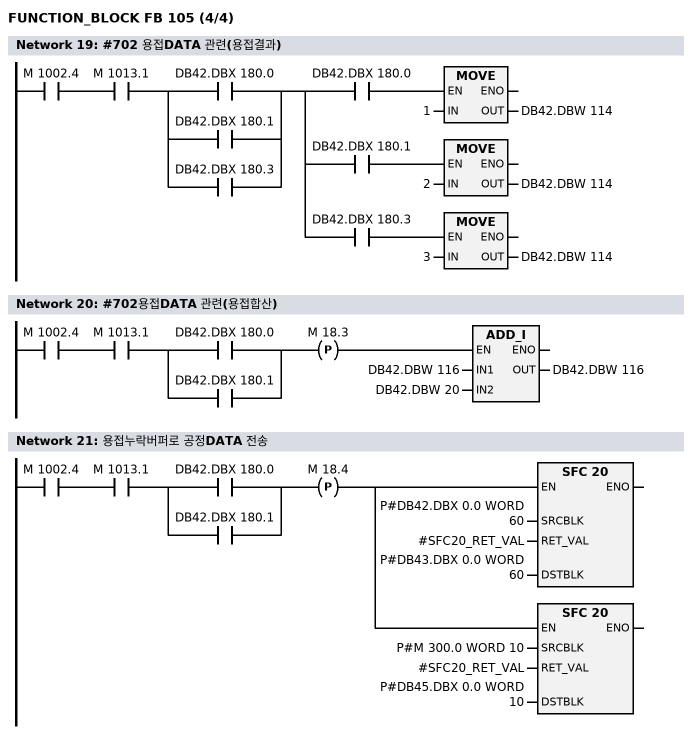

      A     M   1002.4;
      A     M   1013.1;
      A(    ;
      O     DB42.DBX  180.0;
      O     DB42.DBX  180.1;
      O     DB42.DBX  180.3;
      )     ;
      =     L      2.0;
      A     L      2.0;
      A     DB42.DBX  180.0;
      JNB   _022;
      L     1;
      T     DB42.DBW  114;
_022: NOP   0;
      A     L      2.0;
      A     DB42.DBX  180.1;
      JNB   _023;
      L     2;
      T     DB42.DBW  114;
_023: NOP   0;
      A     L      2.0;
      A     DB42.DBX  180.3;
      JNB   _024;
      L     3;
      T     DB42.DBW  114;
_024: NOP   0;
NETWORK
TITLE =#702용접DATA 관련(용접합산)

      A     M   1002.4;
      A     M   1013.1;
      A(    ;
      O     DB42.DBX  180.0;
      O     DB42.DBX  180.1;
      )     ;
      FP    M     18.3;
      JNB   _025;
      L     DB42.DBW  116;
      L     DB42.DBW   20;
      +I    ;
      T     DB42.DBW  116;
_025: NOP   0;
NETWORK
TITLE =용접누락버퍼로 공정DATA 전송

      A     M   1002.4;
      A     M   1013.1;
      A(    ;
      O     DB42.DBX  180.0;
      O     DB42.DBX  180.1;
      )     ;
      FP    M     18.4;
      =     L      2.0;
      A     L      2.0;
      JNB   _026;
      CALL SFC   20 (
           SRCBLK                   := P#DB42.DBX 0.0 WORD 60,
           RET_VAL                  := #SFC20_RET_VAL,
           DSTBLK                   := P#DB43.DBX 0.0 WORD 60);
_026: NOP   0;
      A     L      2.0;
      JNB   _027;
      CALL SFC   20 (
           SRCBLK                   := P#M 300.0 WORD 10,
           RET_VAL                  := #SFC20_RET_VAL,
           DSTBLK                   := P#DB45.DBX 0.0 WORD 10);
_027: NOP   0;
NETWORK
TITLE =용접누락버퍼로 공정DATA 전송

      A     M    501.0;
      FP    M     18.5;
      =     L      2.0;
      A(    ;
      A     L      2.0;
      JNB   _028;
      CALL SFC   20 (
           SRCBLK                   := P#DB43.DBX 960.0 WORD 60,
           RET_VAL                  := #SFC20_RET_VAL,
           DSTBLK                   := P#DB43.DBX 1080.0 WORD 60);
_028: A     BR;
      )     ;
      JNB   _029;
      CALL SFC   20 (
           SRCBLK                   := P#DB43.DBX 840.0 WORD 60,
           RET_VAL                  := #SFC20_RET_VAL,
           DSTBLK                   := P#DB43.DBX 960.0 WORD 60);
_029: NOP   0;
      A(    ;
      A     L      2.0;
      JNB   _02a;
      CALL SFC   20 (
           SRCBLK                   := P#DB43.DBX 720.0 WORD 60,
           RET_VAL                  := #SFC20_RET_VAL,
           DSTBLK                   := P#DB43.DBX 840.0 WORD 60);
_02a: A     BR;
      )     ;
      JNB   _02b;
      CALL SFC   20 (
           SRCBLK                   := P#DB43.DBX 600.0 WORD 60,
           RET_VAL                  := #SFC20_RET_VAL,
           DSTBLK                   := P#DB43.DBX 720.0 WORD 60);
_02b: NOP   0;
      A(    ;
      A     L      2.0;
      JNB   _02c;
      CALL SFC   20 (
           SRCBLK                   := P#DB43.DBX 480.0 WORD 60,
           RET_VAL                  := #SFC20_RET_VAL,
           DSTBLK                   := P#DB43.DBX 600.0 WORD 60);
_02c: A     BR;
      )     ;
      JNB   _02d;
      CALL SFC   20 (
           SRCBLK                   := P#DB43.DBX 360.0 WORD 60,
           RET_VAL                  := #SFC20_RET_VAL,
           DSTBLK                   := P#DB43.DBX 480.0 WORD 60);
_02d: NOP   0;
      A(    ;
      A     L      2.0;
      JNB   _02e;
      CALL SFC   20 (
           SRCBLK                   := P#DB43.DBX 240.0 WORD 60,
           RET_VAL                  := #SFC20_RET_VAL,
           DSTBLK                   := P#DB43.DBX 360.0 WORD 60);
_02e: A     BR;
      )     ;
      JNB   _02f;
      CALL SFC   20 (
           SRCBLK                   := P#DB43.DBX 120.0 WORD 60,
           RET_VAL                  := #SFC20_RET_VAL,
           DSTBLK                   := P#DB43.DBX 240.0 WORD 60);
_02f: NOP   0;
      A     L      2.0;
      JNB   _030;
      CALL SFC   20 (
           SRCBLK                   := P#DB43.DBX 0.0 WORD 60,
           RET_VAL                  := #SFC20_RET_VAL,
           DSTBLK                   := P#DB43.DBX 120.0 WORD 60);
_030: NOP   0;
      A     L      2.0;
      JNB   _031;
      CALL SFC   21 (
           BVAL                     := P#M 40.0 WORD 1,
           RET_VAL                  := #SFC20_RET_VAL,
           BLK                      := P#DB43.DBX 0.0 WORD 60);
_031: NOP   0;
      A(    ;
      A     L      2.0;
      JNB   _032;
      CALL SFC   20 (
           SRCBLK                   := P#DB45.DBX 160.0 WORD 10,
           RET_VAL                  := #SFC20_RET_VAL,
           DSTBLK                   := P#DB45.DBX 180.0 WORD 10);
_032: A     BR;
      )     ;
      JNB   _033;
      CALL SFC   20 (
           SRCBLK                   := P#DB45.DBX 140.0 WORD 10,
           RET_VAL                  := #SFC20_RET_VAL,
           DSTBLK                   := P#DB45.DBX 160.0 WORD 10);
_033: NOP   0;
      A(    ;
      A     L      2.0;
      JNB   _034;
      CALL SFC   20 (
           SRCBLK                   := P#DB45.DBX 120.0 WORD 10,
           RET_VAL                  := #SFC20_RET_VAL,
           DSTBLK                   := P#DB45.DBX 140.0 WORD 10);
_034: A     BR;
      )     ;
      JNB   _035;
      CALL SFC   20 (
           SRCBLK                   := P#DB45.DBX 100.0 WORD 10,
           RET_VAL                  := #SFC20_RET_VAL,
           DSTBLK                   := P#DB45.DBX 120.0 WORD 10);
_035: NOP   0;
      A(    ;
      A     L      2.0;
      JNB   _036;
      CALL SFC   20 (
           SRCBLK                   := P#DB45.DBX 80.0 WORD 10,
           RET_VAL                  := #SFC20_RET_VAL,
           DSTBLK                   := P#DB45.DBX 100.0 WORD 10);
_036: A     BR;
      )     ;
      JNB   _037;
      CALL SFC   20 (
           SRCBLK                   := P#DB45.DBX 60.0 WORD 10,
           RET_VAL                  := #SFC20_RET_VAL,
           DSTBLK                   := P#DB45.DBX 80.0 WORD 10);
_037: NOP   0;
      A(    ;
      A     L      2.0;
      JNB   _038;
      CALL SFC   20 (
           SRCBLK                   := P#DB45.DBX 40.0 WORD 10,
           RET_VAL                  := #SFC20_RET_VAL,
           DSTBLK                   := P#DB45.DBX 60.0 WORD 10);
_038: A     BR;
      )     ;
      JNB   _039;
      CALL SFC   20 (
           SRCBLK                   := P#DB45.DBX 20.0 WORD 10,
           RET_VAL                  := #SFC20_RET_VAL,
           DSTBLK                   := P#DB45.DBX 40.0 WORD 10);
_039: NOP   0;
      A     L      2.0;
      JNB   _03a;
      CALL SFC   20 (
           SRCBLK                   := P#DB45.DBX 0.0 WORD 10,
           RET_VAL                  := #SFC20_RET_VAL,
           DSTBLK                   := P#DB45.DBX 20.0 WORD 10);
_03a: NOP   0;
      A     L      2.0;
      JNB   _03b;
      CALL SFC   21 (
           BVAL                     := P#M 40.0 WORD 1,
           RET_VAL                  := #SFC20_RET_VAL,
           BLK                      := P#DB45.DBX 0.0 WORD 10);
_03b: NOP   0;
NETWORK
TITLE =용접누락버퍼로 공정DATA 전송
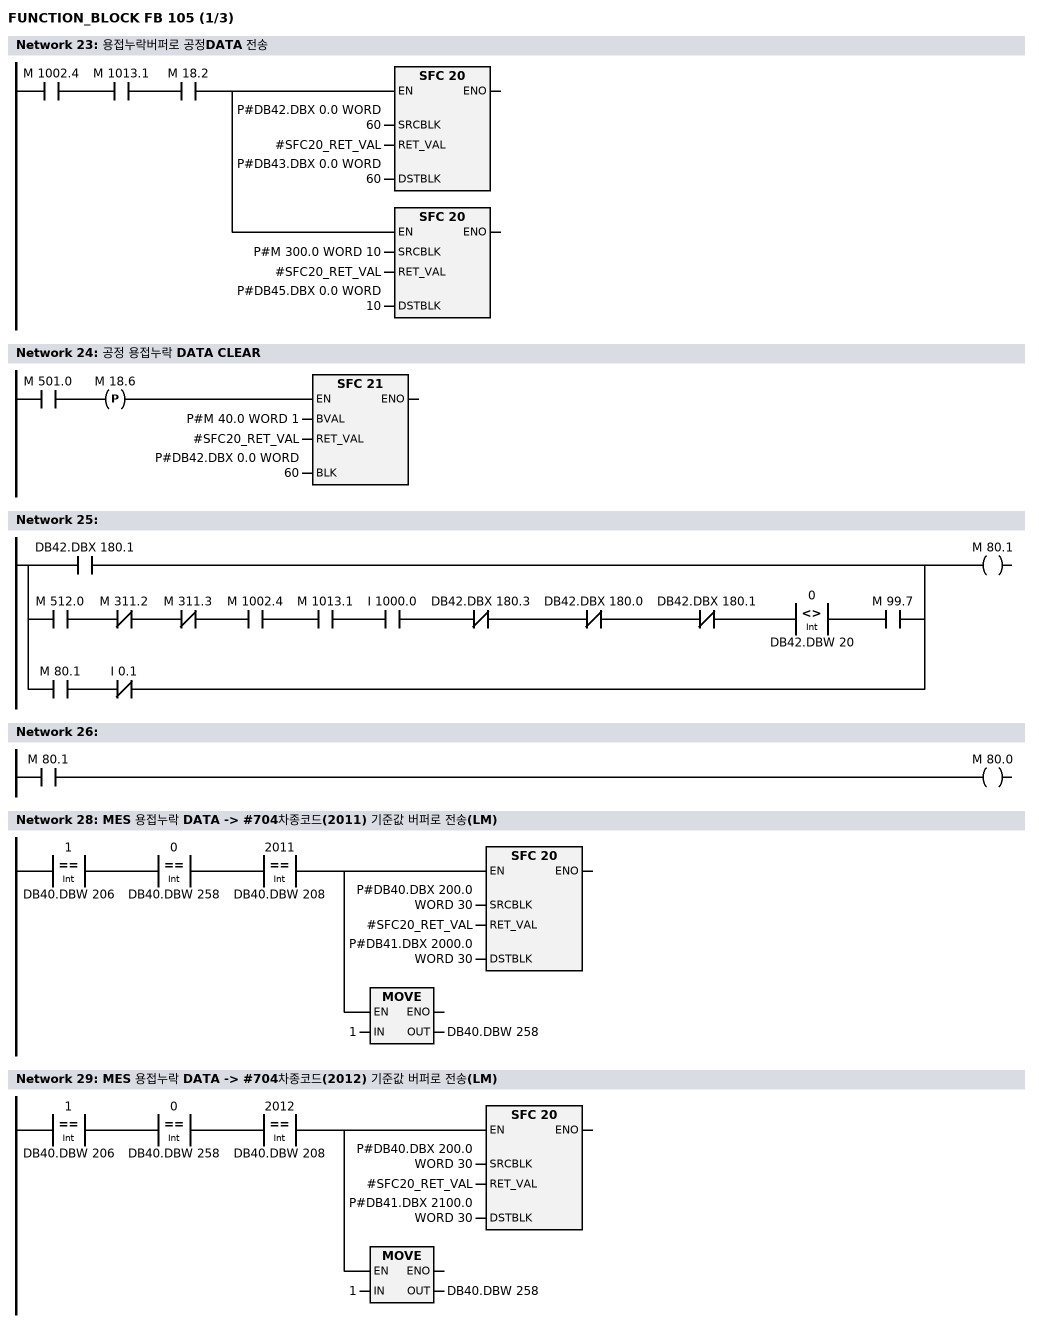

      A     M   1002.4;
      A     M   1013.1;
      A     M     18.2;
      =     L      2.0;
      A     L      2.0;
      JNB   _03c;
      CALL SFC   20 (
           SRCBLK                   := P#DB42.DBX 0.0 WORD 60,
           RET_VAL                  := #SFC20_RET_VAL,
           DSTBLK                   := P#DB43.DBX 0.0 WORD 60);
_03c: NOP   0;
      A     L      2.0;
      JNB   _03d;
      CALL SFC   20 (
           SRCBLK                   := P#M 300.0 WORD 10,
           RET_VAL                  := #SFC20_RET_VAL,
           DSTBLK                   := P#DB45.DBX 0.0 WORD 10);
_03d: NOP   0;
NETWORK
TITLE =공정 용접누락 DATA CLEAR

      A     M    501.0;
      FP    M     18.6;
      JNB   _03e;
      CALL SFC   21 (
           BVAL                     := P#M 40.0 WORD 1,
           RET_VAL                  := #SFC20_RET_VAL,
           BLK                      := P#DB42.DBX 0.0 WORD 60);
_03e: NOP   0;
NETWORK
TITLE =

      O     DB42.DBX  180.1;
      O     ;
      A     M    512.0;
      AN    M    311.2;
      AN    M    311.3;
      A     M   1002.4;
      A     M   1013.1;
      A     I   1000.0;
      AN    DB42.DBX  180.3;
      AN    DB42.DBX  180.0;
      AN    DB42.DBX  180.1;
      A(    ;
      L     0;
      L     DB42.DBW   20;
      <>I   ;
      )     ;
      A     M     99.7;
      O     ;
      A     M     80.1;
      AN    I      0.1;
      =     M     80.1;
NETWORK
TITLE =

      A     M     80.1;
      =     M     80.0;
NETWORK
TITLE =

NETWORK
TITLE =MES 용접누락 DATA -> #704차종코드(2011) 기준값 버퍼로 전송(LM)

      A(    ;
      L     1;
      L     DB40.DBW  206;
      ==I   ;
      )     ;
      A(    ;
      L     0;
      L     DB40.DBW  258;
      ==I   ;
      )     ;
      A(    ;
      L     2011;
      L     DB40.DBW  208;
      ==I   ;
      )     ;
      =     L      2.0;
      A     L      2.0;
      JNB   _03f;
      CALL SFC   20 (
           SRCBLK                   := P#DB40.DBX 200.0 WORD 30,
           RET_VAL                  := #SFC20_RET_VAL,
           DSTBLK                   := P#DB41.DBX 2000.0 WORD 30);
_03f: NOP   0;
      A     L      2.0;
      JNB   _040;
      L     1;
      T     DB40.DBW  258;
_040: NOP   0;
NETWORK
TITLE =MES 용접누락 DATA -> #704차종코드(2012) 기준값 버퍼로 전송(LM)

      A(    ;
      L     1;
      L     DB40.DBW  206;
      ==I   ;
      )     ;
      A(    ;
      L     0;
      L     DB40.DBW  258;
      ==I   ;
      )     ;
      A(    ;
      L     2012;
      L     DB40.DBW  208;
      ==I   ;
      )     ;
      =     L      2.0;
      A     L      2.0;
      JNB   _041;
      CALL SFC   20 (
           SRCBLK                   := P#DB40.DBX 200.0 WORD 30,
           RET_VAL                  := #SFC20_RET_VAL,
           DSTBLK                   := P#DB41.DBX 2100.0 WORD 30);
_041: NOP   0;
      A     L      2.0;
      JNB   _042;
      L     1;
      T     DB40.DBW  258;
_042: NOP   0;
NETWORK
TITLE =MES 용접누락 DATA -> #704차종코드(2013) 기준값 버퍼로 전송(LM)
//
//
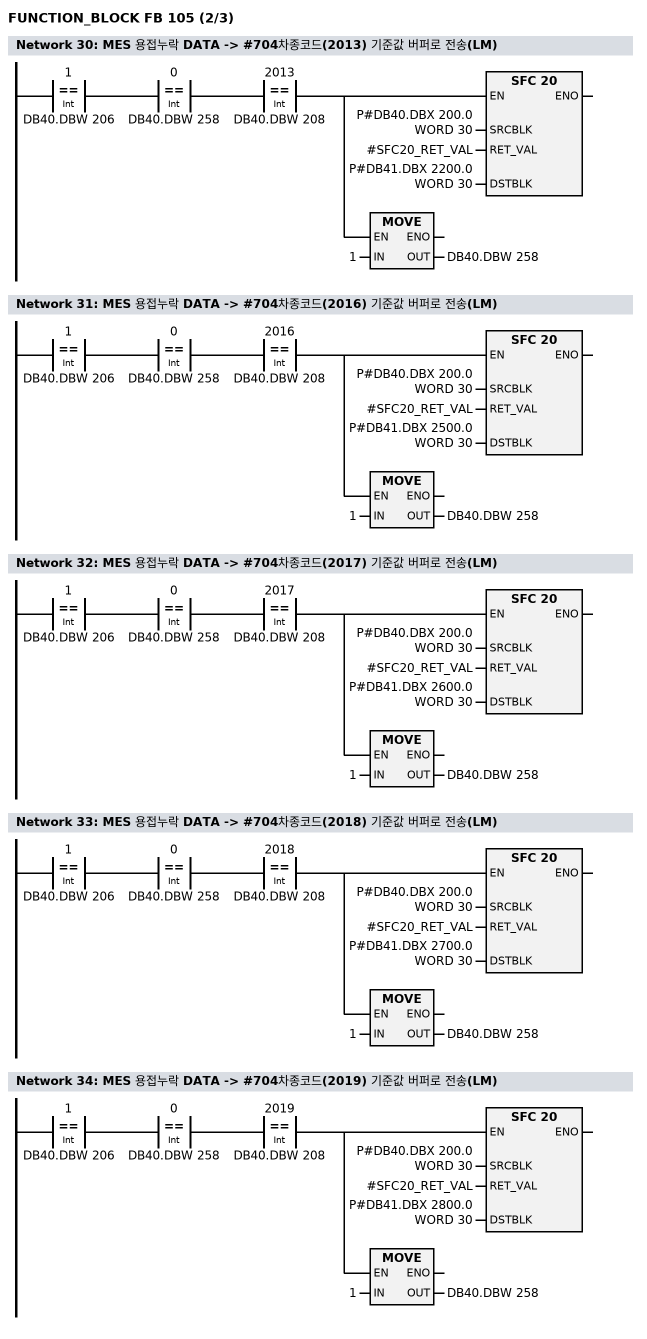
      A(    ;
      L     1;
      L     DB40.DBW  206;
      ==I   ;
      )     ;
      A(    ;
      L     0;
      L     DB40.DBW  258;
      ==I   ;
      )     ;
      A(    ;
      L     2013;
      L     DB40.DBW  208;
      ==I   ;
      )     ;
      =     L      2.0;
      A     L      2.0;
      JNB   _043;
      CALL SFC   20 (
           SRCBLK                   := P#DB40.DBX 200.0 WORD 30,
           RET_VAL                  := #SFC20_RET_VAL,
           DSTBLK                   := P#DB41.DBX 2200.0 WORD 30);
_043: NOP   0;
      A     L      2.0;
      JNB   _044;
      L     1;
      T     DB40.DBW  258;
_044: NOP   0;
NETWORK
TITLE =MES 용접누락 DATA -> #704차종코드(2016) 기준값 버퍼로 전송(LM)

      A(    ;
      L     1;
      L     DB40.DBW  206;
      ==I   ;
      )     ;
      A(    ;
      L     0;
      L     DB40.DBW  258;
      ==I   ;
      )     ;
      A(    ;
      L     2016;
      L     DB40.DBW  208;
      ==I   ;
      )     ;
      =     L      2.0;
      A     L      2.0;
      JNB   _045;
      CALL SFC   20 (
           SRCBLK                   := P#DB40.DBX 200.0 WORD 30,
           RET_VAL                  := #SFC20_RET_VAL,
           DSTBLK                   := P#DB41.DBX 2500.0 WORD 30);
_045: NOP   0;
      A     L      2.0;
      JNB   _046;
      L     1;
      T     DB40.DBW  258;
_046: NOP   0;
NETWORK
TITLE =MES 용접누락 DATA -> #704차종코드(2017) 기준값 버퍼로 전송(LM)

      A(    ;
      L     1;
      L     DB40.DBW  206;
      ==I   ;
      )     ;
      A(    ;
      L     0;
      L     DB40.DBW  258;
      ==I   ;
      )     ;
      A(    ;
      L     2017;
      L     DB40.DBW  208;
      ==I   ;
      )     ;
      =     L      2.0;
      A     L      2.0;
      JNB   _047;
      CALL SFC   20 (
           SRCBLK                   := P#DB40.DBX 200.0 WORD 30,
           RET_VAL                  := #SFC20_RET_VAL,
           DSTBLK                   := P#DB41.DBX 2600.0 WORD 30);
_047: NOP   0;
      A     L      2.0;
      JNB   _048;
      L     1;
      T     DB40.DBW  258;
_048: NOP   0;
NETWORK
TITLE =MES 용접누락 DATA -> #704차종코드(2018) 기준값 버퍼로 전송(LM)

      A(    ;
      L     1;
      L     DB40.DBW  206;
      ==I   ;
      )     ;
      A(    ;
      L     0;
      L     DB40.DBW  258;
      ==I   ;
      )     ;
      A(    ;
      L     2018;
      L     DB40.DBW  208;
      ==I   ;
      )     ;
      =     L      2.0;
      A     L      2.0;
      JNB   _049;
      CALL SFC   20 (
           SRCBLK                   := P#DB40.DBX 200.0 WORD 30,
           RET_VAL                  := #SFC20_RET_VAL,
           DSTBLK                   := P#DB41.DBX 2700.0 WORD 30);
_049: NOP   0;
      A     L      2.0;
      JNB   _04a;
      L     1;
      T     DB40.DBW  258;
_04a: NOP   0;
NETWORK
TITLE =MES 용접누락 DATA -> #704차종코드(2019) 기준값 버퍼로 전송(LM)

      A(    ;
      L     1;
      L     DB40.DBW  206;
      ==I   ;
      )     ;
      A(    ;
      L     0;
      L     DB40.DBW  258;
      ==I   ;
      )     ;
      A(    ;
      L     2019;
      L     DB40.DBW  208;
      ==I   ;
      )     ;
      =     L      2.0;
      A     L      2.0;
      JNB   _04b;
      CALL SFC   20 (
           SRCBLK                   := P#DB40.DBX 200.0 WORD 30,
           RET_VAL                  := #SFC20_RET_VAL,
           DSTBLK                   := P#DB41.DBX 2800.0 WORD 30);
_04b: NOP   0;
      A     L      2.0;
      JNB   _04c;
      L     1;
      T     DB40.DBW  258;
_04c: NOP   0;
NETWORK
TITLE =MES 용접누락 DATA -> #704차종코드(2101) 기준값 버퍼로 전송(TL)
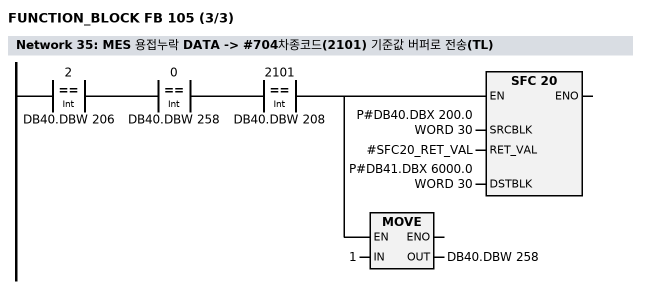

      A(    ;
      L     2;
      L     DB40.DBW  206;
      ==I   ;
      )     ;
      A(    ;
      L     0;
      L     DB40.DBW  258;
      ==I   ;
      )     ;
      A(    ;
      L     2101;
      L     DB40.DBW  208;
      ==I   ;
      )     ;
      =     L      2.0;
      A     L      2.0;
      JNB   _04d;
      CALL SFC   20 (
           SRCBLK                   := P#DB40.DBX 200.0 WORD 30,
           RET_VAL                  := #SFC20_RET_VAL,
           DSTBLK                   := P#DB41.DBX 6000.0 WORD 30);
_04d: NOP   0;
      A     L      2.0;
      JNB   _04e;
      L     1;
      T     DB40.DBW  258;
_04e: NOP   0;
NETWORK
TITLE =#704 RBT1호 용접카운터 INT -> DB로 전송보조

      AN    OV;
      =     L      2.0;
      A     L      2.0;
      A     I   1012.0;
      =     M     21.0;
      A     L      2.0;
      A     I   1012.1;
      =     M     21.1;
      A     L      2.0;
      A     I   1012.2;
      =     M     21.2;
      A     L      2.0;
      A     I   1012.3;
      =     M     21.3;
      A     L      2.0;
      A     I   1012.4;
      =     M     21.4;
      A     L      2.0;
      AN    M      3.3;
      =     L      2.1;
      A     L      2.1;
      A     I   1012.5;
      =     M     21.5;
      A     L      2.1;
      A     I   1012.6;
      =     M     21.6;
      A     L      2.1;
      A     I   1012.7;
      =     M     21.7;
NETWORK
TITLE =#704 RBT1호 용접카운터 INT -> DB로 전송
//
//
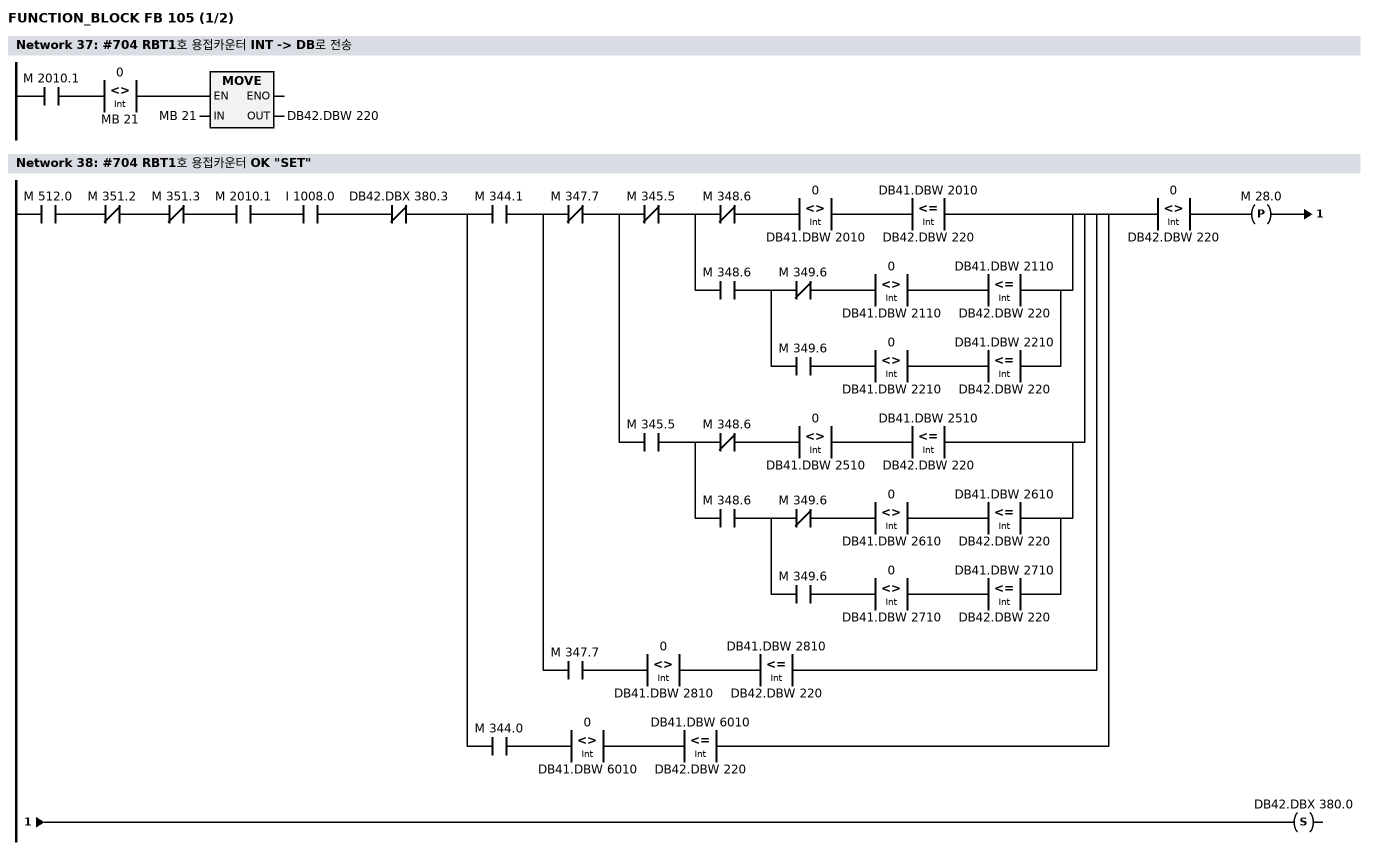
      A     M   2010.1;
      A(    ;
      L     0;
      L     MB    21;
      <>I   ;
      )     ;
      JNB   _04f;
      L     MB    21;
      T     DB42.DBW  220;
_04f: NOP   0;
NETWORK
TITLE =#704 RBT1호 용접카운터 OK "SET"

      A     M    512.0;
      AN    M    351.2;
      AN    M    351.3;
      A     M   2010.1;
      A     I   1008.0;
      AN    DB42.DBX  380.3;
      A(    ;
      A     M    344.1;
      A(    ;
      AN    M    347.7;
      A(    ;
      AN    M    345.5;
      A(    ;
      AN    M    348.6;
      A(    ;
      L     0;
      L     DB41.DBW 2010;
      <>I   ;
      )     ;
      A(    ;
      L     DB41.DBW 2010;
      L     DB42.DBW  220;
      <=I   ;
      )     ;
      O     ;
      A     M    348.6;
      A(    ;
      AN    M    349.6;
      A(    ;
      L     0;
      L     DB41.DBW 2110;
      <>I   ;
      )     ;
      A(    ;
      L     DB41.DBW 2110;
      L     DB42.DBW  220;
      <=I   ;
      )     ;
      O     ;
      A     M    349.6;
      A(    ;
      L     0;
      L     DB41.DBW 2210;
      <>I   ;
      )     ;
      A(    ;
      L     DB41.DBW 2210;
      L     DB42.DBW  220;
      <=I   ;
      )     ;
      )     ;
      )     ;
      O     ;
      A     M    345.5;
      A(    ;
      AN    M    348.6;
      A(    ;
      L     0;
      L     DB41.DBW 2510;
      <>I   ;
      )     ;
      A(    ;
      L     DB41.DBW 2510;
      L     DB42.DBW  220;
      <=I   ;
      )     ;
      O     ;
      A     M    348.6;
      A(    ;
      AN    M    349.6;
      A(    ;
      L     0;
      L     DB41.DBW 2610;
      <>I   ;
      )     ;
      A(    ;
      L     DB41.DBW 2610;
      L     DB42.DBW  220;
      <=I   ;
      )     ;
      O     ;
      A     M    349.6;
      A(    ;
      L     0;
      L     DB41.DBW 2710;
      <>I   ;
      )     ;
      A(    ;
      L     DB41.DBW 2710;
      L     DB42.DBW  220;
      <=I   ;
      )     ;
      )     ;
      )     ;
      )     ;
      O     ;
      A     M    347.7;
      A(    ;
      L     0;
      L     DB41.DBW 2810;
      <>I   ;
      )     ;
      A(    ;
      L     DB41.DBW 2810;
      L     DB42.DBW  220;
      <=I   ;
      )     ;
      )     ;
      O     ;
      A     M    344.0;
      A(    ;
      L     0;
      L     DB41.DBW 6010;
      <>I   ;
      )     ;
      A(    ;
      L     DB41.DBW 6010;
      L     DB42.DBW  220;
      <=I   ;
      )     ;
      )     ;
      A(    ;
      L     0;
      L     DB42.DBW  220;
      <>I   ;
      )     ;
      FP    M     28.0;
      S     DB42.DBX  380.0;
NETWORK
TITLE =#704 RBT1호 용접카운터 NG "SET"
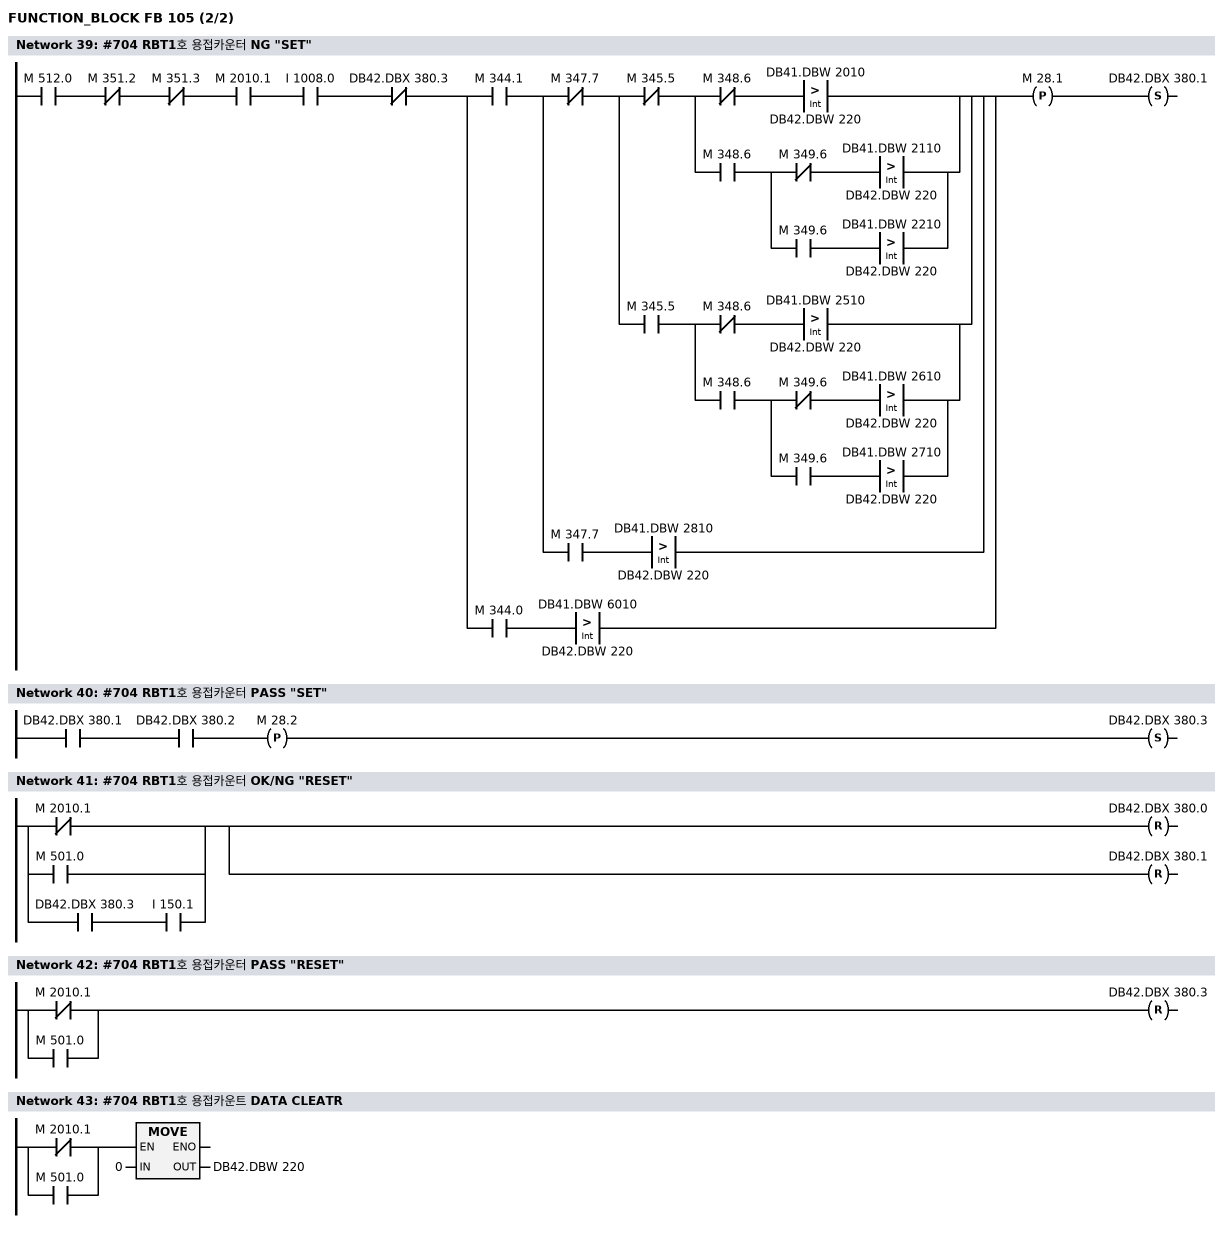

      A     M    512.0;
      AN    M    351.2;
      AN    M    351.3;
      A     M   2010.1;
      A     I   1008.0;
      AN    DB42.DBX  380.3;
      A(    ;
      A     M    344.1;
      A(    ;
      AN    M    347.7;
      A(    ;
      AN    M    345.5;
      A(    ;
      AN    M    348.6;
      A(    ;
      L     DB41.DBW 2010;
      L     DB42.DBW  220;
      >I    ;
      )     ;
      O     ;
      A     M    348.6;
      A(    ;
      AN    M    349.6;
      A(    ;
      L     DB41.DBW 2110;
      L     DB42.DBW  220;
      >I    ;
      )     ;
      O     ;
      A     M    349.6;
      A(    ;
      L     DB41.DBW 2210;
      L     DB42.DBW  220;
      >I    ;
      )     ;
      )     ;
      )     ;
      O     ;
      A     M    345.5;
      A(    ;
      AN    M    348.6;
      A(    ;
      L     DB41.DBW 2510;
      L     DB42.DBW  220;
      >I    ;
      )     ;
      O     ;
      A     M    348.6;
      A(    ;
      AN    M    349.6;
      A(    ;
      L     DB41.DBW 2610;
      L     DB42.DBW  220;
      >I    ;
      )     ;
      O     ;
      A     M    349.6;
      A(    ;
      L     DB41.DBW 2710;
      L     DB42.DBW  220;
      >I    ;
      )     ;
      )     ;
      )     ;
      )     ;
      O     ;
      A     M    347.7;
      A(    ;
      L     DB41.DBW 2810;
      L     DB42.DBW  220;
      >I    ;
      )     ;
      )     ;
      O     ;
      A     M    344.0;
      A(    ;
      L     DB41.DBW 6010;
      L     DB42.DBW  220;
      >I    ;
      )     ;
      )     ;
      FP    M     28.1;
      S     DB42.DBX  380.1;
NETWORK
TITLE =#704 RBT1호 용접카운터 PASS "SET"

      A     DB42.DBX  380.1;
      A     DB42.DBX  380.2;
      FP    M     28.2;
      S     DB42.DBX  380.3;
NETWORK
TITLE =#704 RBT1호 용접카운터 OK/NG "RESET"

      ON    M   2010.1;
      O     M    501.0;
      O     ;
      A     DB42.DBX  380.3;
      A     I    150.1;
      R     DB42.DBX  380.0;
      R     DB42.DBX  380.1;
NETWORK
TITLE =#704 RBT1호 용접카운터 PASS "RESET"

      ON    M   2010.1;
      O     M    501.0;
      R     DB42.DBX  380.3;
NETWORK
TITLE =#704 RBT1호 용접카운트 DATA CLEATR

      A(    ;
      ON    M   2010.1;
      O     M    501.0;
      )     ;
      JNB   _050;
      L     0;
      T     DB42.DBW  220;
_050: NOP   0;
NETWORK
TITLE =#704 RBT2호 용접카운터 INT -> DB로 전송보조

      AN    OV;
      =     L      2.0;
      A     L      2.0;
      A     I   1020.0;
      =     M     22.0;
      A     L      2.0;
      A     I   1020.1;
      =     M     22.1;
      A     L      2.0;
      A     I   1020.2;
      =     M     22.2;
      A     L      2.0;
      A     I   1020.3;
      =     M     22.3;
      A     L      2.0;
      A     I   1020.4;
      =     M     22.4;
      A     L      2.0;
      AN    M      3.3;
      =     L      2.1;
      A     L      2.1;
      A     I   1020.5;
      =     M     22.5;
      A     L      2.1;
      A     I   1020.6;
      =     M     22.6;
      A     L      2.1;
      A     I   1020.7;
      =     M     22.7;
NETWORK
TITLE =#704 RBT2호 용접카운터 INT -> DB로 전송
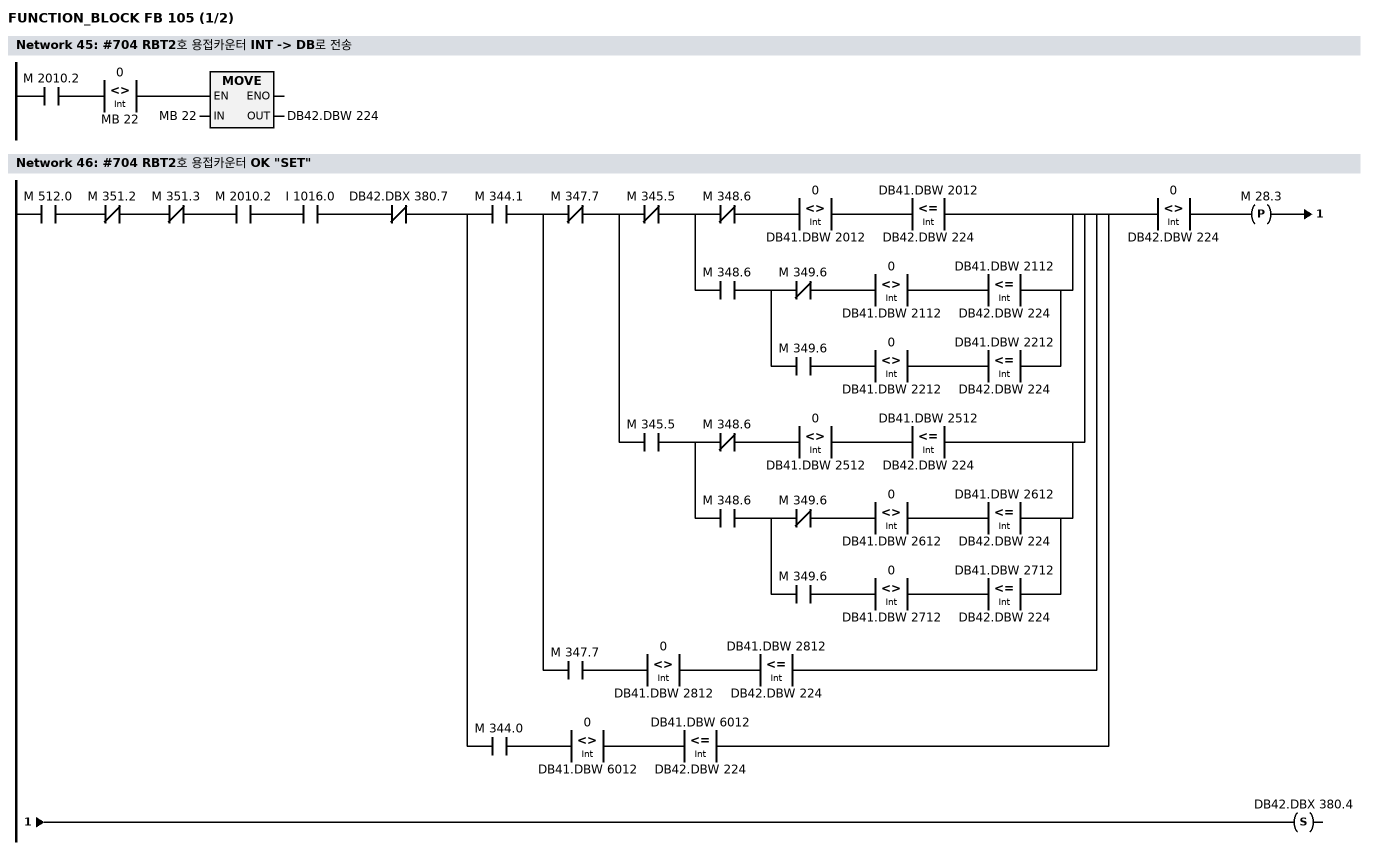

      A     M   2010.2;
      A(    ;
      L     0;
      L     MB    22;
      <>I   ;
      )     ;
      JNB   _051;
      L     MB    22;
      T     DB42.DBW  224;
_051: NOP   0;
NETWORK
TITLE =#704 RBT2호 용접카운터 OK "SET"

      A     M    512.0;
      AN    M    351.2;
      AN    M    351.3;
      A     M   2010.2;
      A     I   1016.0;
      AN    DB42.DBX  380.7;
      A(    ;
      A     M    344.1;
      A(    ;
      AN    M    347.7;
      A(    ;
      AN    M    345.5;
      A(    ;
      AN    M    348.6;
      A(    ;
      L     0;
      L     DB41.DBW 2012;
      <>I   ;
      )     ;
      A(    ;
      L     DB41.DBW 2012;
      L     DB42.DBW  224;
      <=I   ;
      )     ;
      O     ;
      A     M    348.6;
      A(    ;
      AN    M    349.6;
      A(    ;
      L     0;
      L     DB41.DBW 2112;
      <>I   ;
      )     ;
      A(    ;
      L     DB41.DBW 2112;
      L     DB42.DBW  224;
      <=I   ;
      )     ;
      O     ;
      A     M    349.6;
      A(    ;
      L     0;
      L     DB41.DBW 2212;
      <>I   ;
      )     ;
      A(    ;
      L     DB41.DBW 2212;
      L     DB42.DBW  224;
      <=I   ;
      )     ;
      )     ;
      )     ;
      O     ;
      A     M    345.5;
      A(    ;
      AN    M    348.6;
      A(    ;
      L     0;
      L     DB41.DBW 2512;
      <>I   ;
      )     ;
      A(    ;
      L     DB41.DBW 2512;
      L     DB42.DBW  224;
      <=I   ;
      )     ;
      O     ;
      A     M    348.6;
      A(    ;
      AN    M    349.6;
      A(    ;
      L     0;
      L     DB41.DBW 2612;
      <>I   ;
      )     ;
      A(    ;
      L     DB41.DBW 2612;
      L     DB42.DBW  224;
      <=I   ;
      )     ;
      O     ;
      A     M    349.6;
      A(    ;
      L     0;
      L     DB41.DBW 2712;
      <>I   ;
      )     ;
      A(    ;
      L     DB41.DBW 2712;
      L     DB42.DBW  224;
      <=I   ;
      )     ;
      )     ;
      )     ;
      )     ;
      O     ;
      A     M    347.7;
      A(    ;
      L     0;
      L     DB41.DBW 2812;
      <>I   ;
      )     ;
      A(    ;
      L     DB41.DBW 2812;
      L     DB42.DBW  224;
      <=I   ;
      )     ;
      )     ;
      O     ;
      A     M    344.0;
      A(    ;
      L     0;
      L     DB41.DBW 6012;
      <>I   ;
      )     ;
      A(    ;
      L     DB41.DBW 6012;
      L     DB42.DBW  224;
      <=I   ;
      )     ;
      )     ;
      A(    ;
      L     0;
      L     DB42.DBW  224;
      <>I   ;
      )     ;
      FP    M     28.3;
      S     DB42.DBX  380.4;
NETWORK
TITLE =#704 RBT2호 용접카운터 NG "SET"
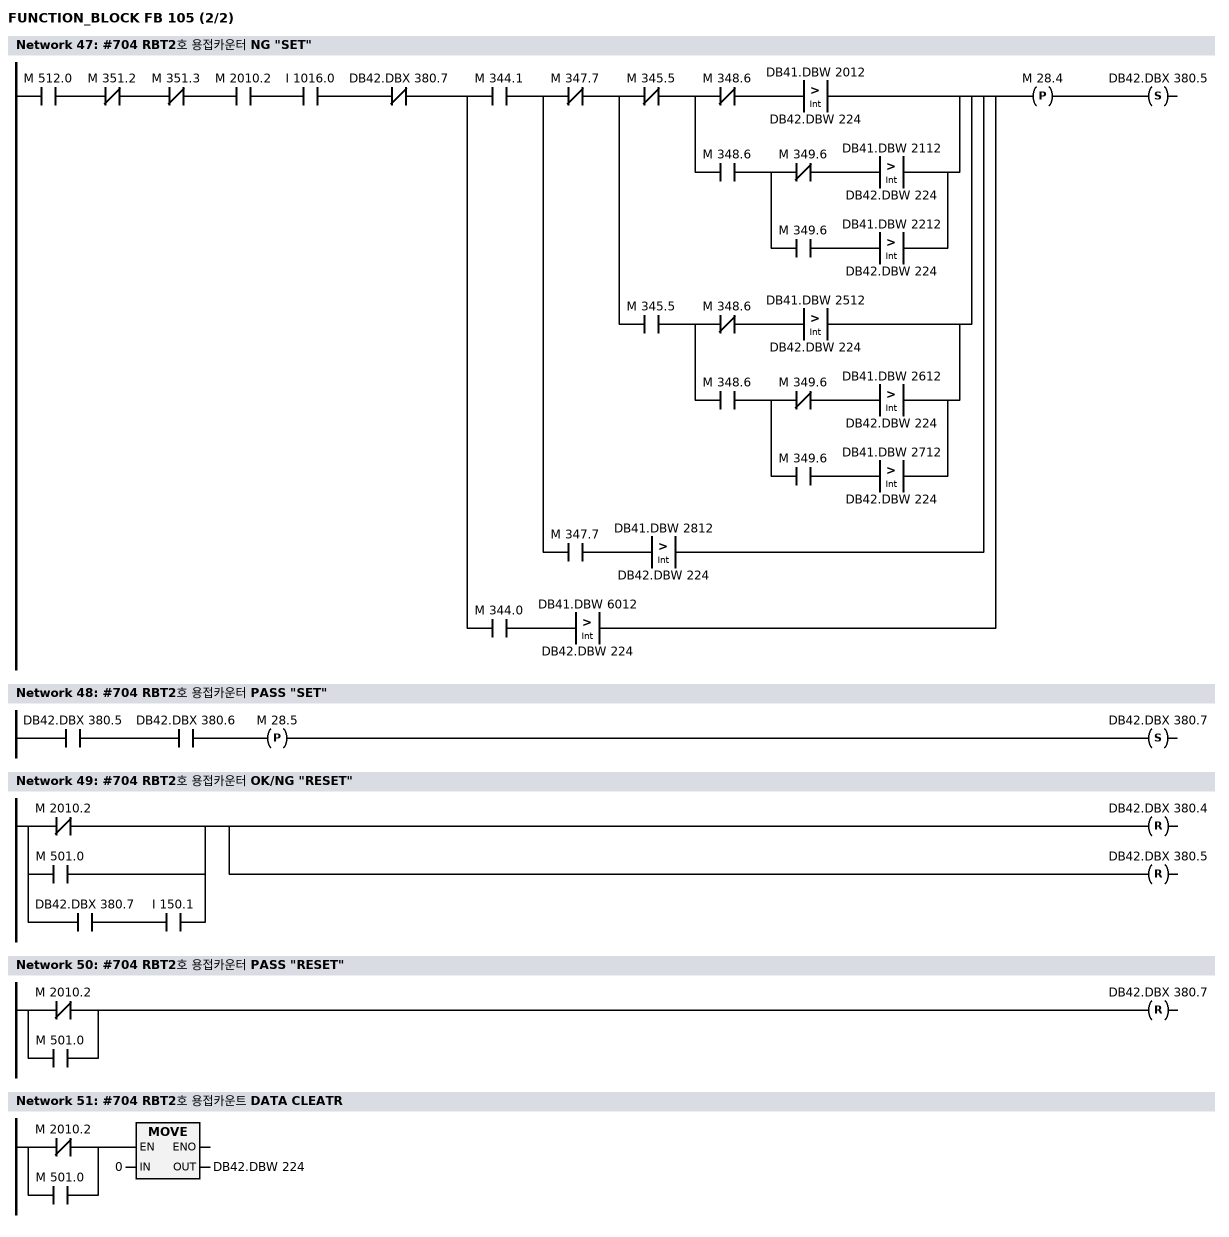

      A     M    512.0;
      AN    M    351.2;
      AN    M    351.3;
      A     M   2010.2;
      A     I   1016.0;
      AN    DB42.DBX  380.7;
      A(    ;
      A     M    344.1;
      A(    ;
      AN    M    347.7;
      A(    ;
      AN    M    345.5;
      A(    ;
      AN    M    348.6;
      A(    ;
      L     DB41.DBW 2012;
      L     DB42.DBW  224;
      >I    ;
      )     ;
      O     ;
      A     M    348.6;
      A(    ;
      AN    M    349.6;
      A(    ;
      L     DB41.DBW 2112;
      L     DB42.DBW  224;
      >I    ;
      )     ;
      O     ;
      A     M    349.6;
      A(    ;
      L     DB41.DBW 2212;
      L     DB42.DBW  224;
      >I    ;
      )     ;
      )     ;
      )     ;
      O     ;
      A     M    345.5;
      A(    ;
      AN    M    348.6;
      A(    ;
      L     DB41.DBW 2512;
      L     DB42.DBW  224;
      >I    ;
      )     ;
      O     ;
      A     M    348.6;
      A(    ;
      AN    M    349.6;
      A(    ;
      L     DB41.DBW 2612;
      L     DB42.DBW  224;
      >I    ;
      )     ;
      O     ;
      A     M    349.6;
      A(    ;
      L     DB41.DBW 2712;
      L     DB42.DBW  224;
      >I    ;
      )     ;
      )     ;
      )     ;
      )     ;
      O     ;
      A     M    347.7;
      A(    ;
      L     DB41.DBW 2812;
      L     DB42.DBW  224;
      >I    ;
      )     ;
      )     ;
      O     ;
      A     M    344.0;
      A(    ;
      L     DB41.DBW 6012;
      L     DB42.DBW  224;
      >I    ;
      )     ;
      )     ;
      FP    M     28.4;
      S     DB42.DBX  380.5;
NETWORK
TITLE =#704 RBT2호 용접카운터 PASS "SET"
//
//
      A     DB42.DBX  380.5;
      A     DB42.DBX  380.6;
      FP    M     28.5;
      S     DB42.DBX  380.7;
NETWORK
TITLE =#704 RBT2호 용접카운터 OK/NG "RESET"

      ON    M   2010.2;
      O     M    501.0;
      O     ;
      A     DB42.DBX  380.7;
      A     I    150.1;
      R     DB42.DBX  380.4;
      R     DB42.DBX  380.5;
NETWORK
TITLE =#704 RBT2호 용접카운터 PASS "RESET"

      ON    M   2010.2;
      O     M    501.0;
      R     DB42.DBX  380.7;
NETWORK
TITLE =#704 RBT2호 용접카운트 DATA CLEATR

      A(    ;
      ON    M   2010.2;
      O     M    501.0;
      )     ;
      JNB   _052;
      L     0;
      T     DB42.DBW  224;
_052: NOP   0;
NETWORK
TITLE =#704 RBT3호 용접카운터 INT -> DB로 전송보조

      AN    OV;
      =     L      2.0;
      A     L      2.0;
      A     I   1028.0;
      =     M     23.0;
      A     L      2.0;
      A     I   1028.1;
      =     M     23.1;
      A     L      2.0;
      A     I   1028.2;
      =     M     23.2;
      A     L      2.0;
      A     I   1028.3;
      =     M     23.3;
      A     L      2.0;
      A     I   1028.4;
      =     M     23.4;
      A     L      2.0;
      AN    M      3.3;
      =     L      2.1;
      A     L      2.1;
      A     I   1028.5;
      =     M     23.5;
      A     L      2.1;
      A     I   1028.6;
      =     M     23.6;
      A     L      2.1;
      A     I   1028.7;
      =     M     23.7;
NETWORK
TITLE =#704 RBT3호 용접카운터 INT -> DB로 전송
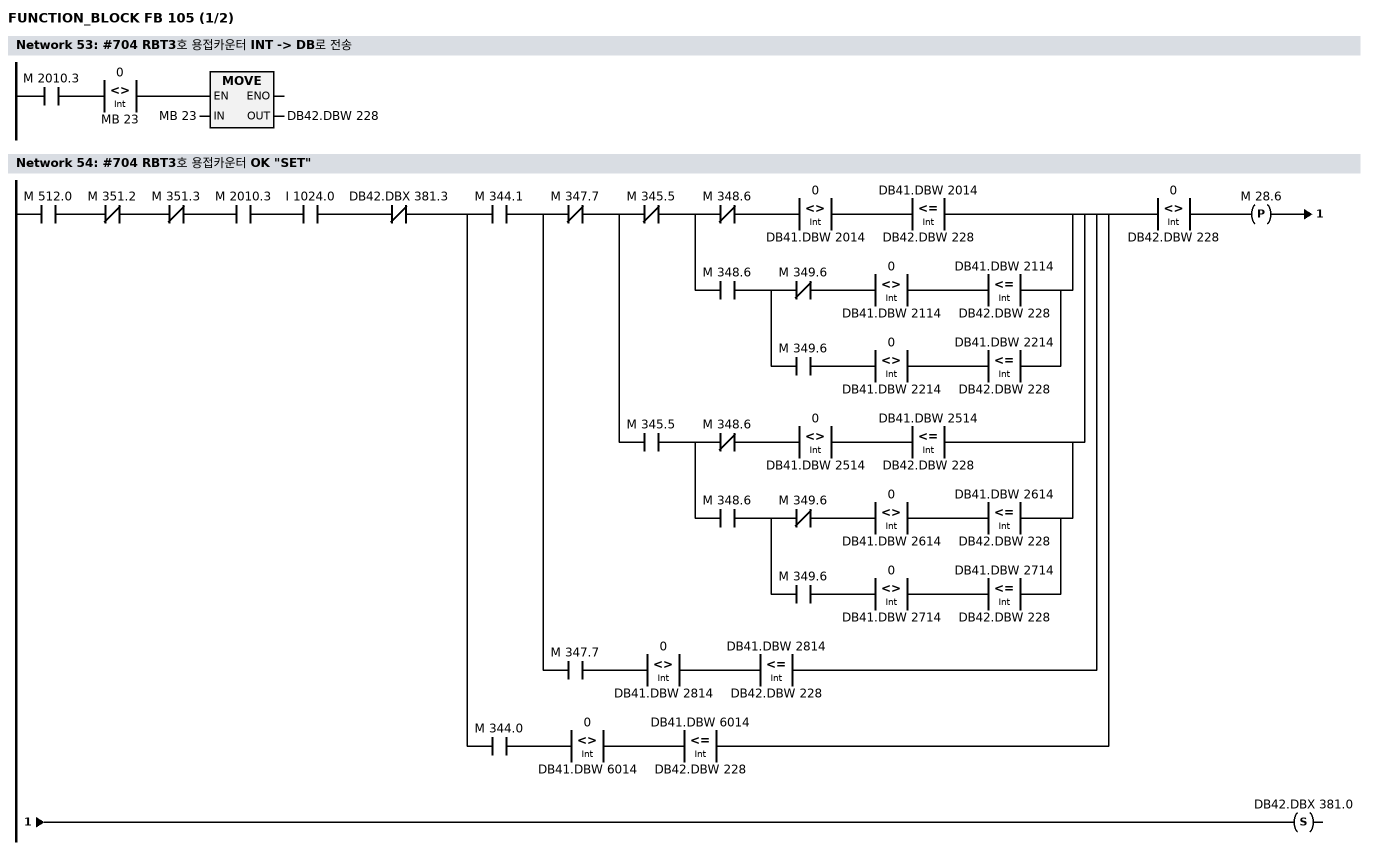

      A     M   2010.3;
      A(    ;
      L     0;
      L     MB    23;
      <>I   ;
      )     ;
      JNB   _053;
      L     MB    23;
      T     DB42.DBW  228;
_053: NOP   0;
NETWORK
TITLE =#704 RBT3호 용접카운터 OK "SET"

      A     M    512.0;
      AN    M    351.2;
      AN    M    351.3;
      A     M   2010.3;
      A     I   1024.0;
      AN    DB42.DBX  381.3;
      A(    ;
      A     M    344.1;
      A(    ;
      AN    M    347.7;
      A(    ;
      AN    M    345.5;
      A(    ;
      AN    M    348.6;
      A(    ;
      L     0;
      L     DB41.DBW 2014;
      <>I   ;
      )     ;
      A(    ;
      L     DB41.DBW 2014;
      L     DB42.DBW  228;
      <=I   ;
      )     ;
      O     ;
      A     M    348.6;
      A(    ;
      AN    M    349.6;
      A(    ;
      L     0;
      L     DB41.DBW 2114;
      <>I   ;
      )     ;
      A(    ;
      L     DB41.DBW 2114;
      L     DB42.DBW  228;
      <=I   ;
      )     ;
      O     ;
      A     M    349.6;
      A(    ;
      L     0;
      L     DB41.DBW 2214;
      <>I   ;
      )     ;
      A(    ;
      L     DB41.DBW 2214;
      L     DB42.DBW  228;
      <=I   ;
      )     ;
      )     ;
      )     ;
      O     ;
      A     M    345.5;
      A(    ;
      AN    M    348.6;
      A(    ;
      L     0;
      L     DB41.DBW 2514;
      <>I   ;
      )     ;
      A(    ;
      L     DB41.DBW 2514;
      L     DB42.DBW  228;
      <=I   ;
      )     ;
      O     ;
      A     M    348.6;
      A(    ;
      AN    M    349.6;
      A(    ;
      L     0;
      L     DB41.DBW 2614;
      <>I   ;
      )     ;
      A(    ;
      L     DB41.DBW 2614;
      L     DB42.DBW  228;
      <=I   ;
      )     ;
      O     ;
      A     M    349.6;
      A(    ;
      L     0;
      L     DB41.DBW 2714;
      <>I   ;
      )     ;
      A(    ;
      L     DB41.DBW 2714;
      L     DB42.DBW  228;
      <=I   ;
      )     ;
      )     ;
      )     ;
      )     ;
      O     ;
      A     M    347.7;
      A(    ;
      L     0;
      L     DB41.DBW 2814;
      <>I   ;
      )     ;
      A(    ;
      L     DB41.DBW 2814;
      L     DB42.DBW  228;
      <=I   ;
      )     ;
      )     ;
      O     ;
      A     M    344.0;
      A(    ;
      L     0;
      L     DB41.DBW 6014;
      <>I   ;
      )     ;
      A(    ;
      L     DB41.DBW 6014;
      L     DB42.DBW  228;
      <=I   ;
      )     ;
      )     ;
      A(    ;
      L     0;
      L     DB42.DBW  228;
      <>I   ;
      )     ;
      FP    M     28.6;
      S     DB42.DBX  381.0;
NETWORK
TITLE =#704 RBT3호 용접카운터 NG "SET"
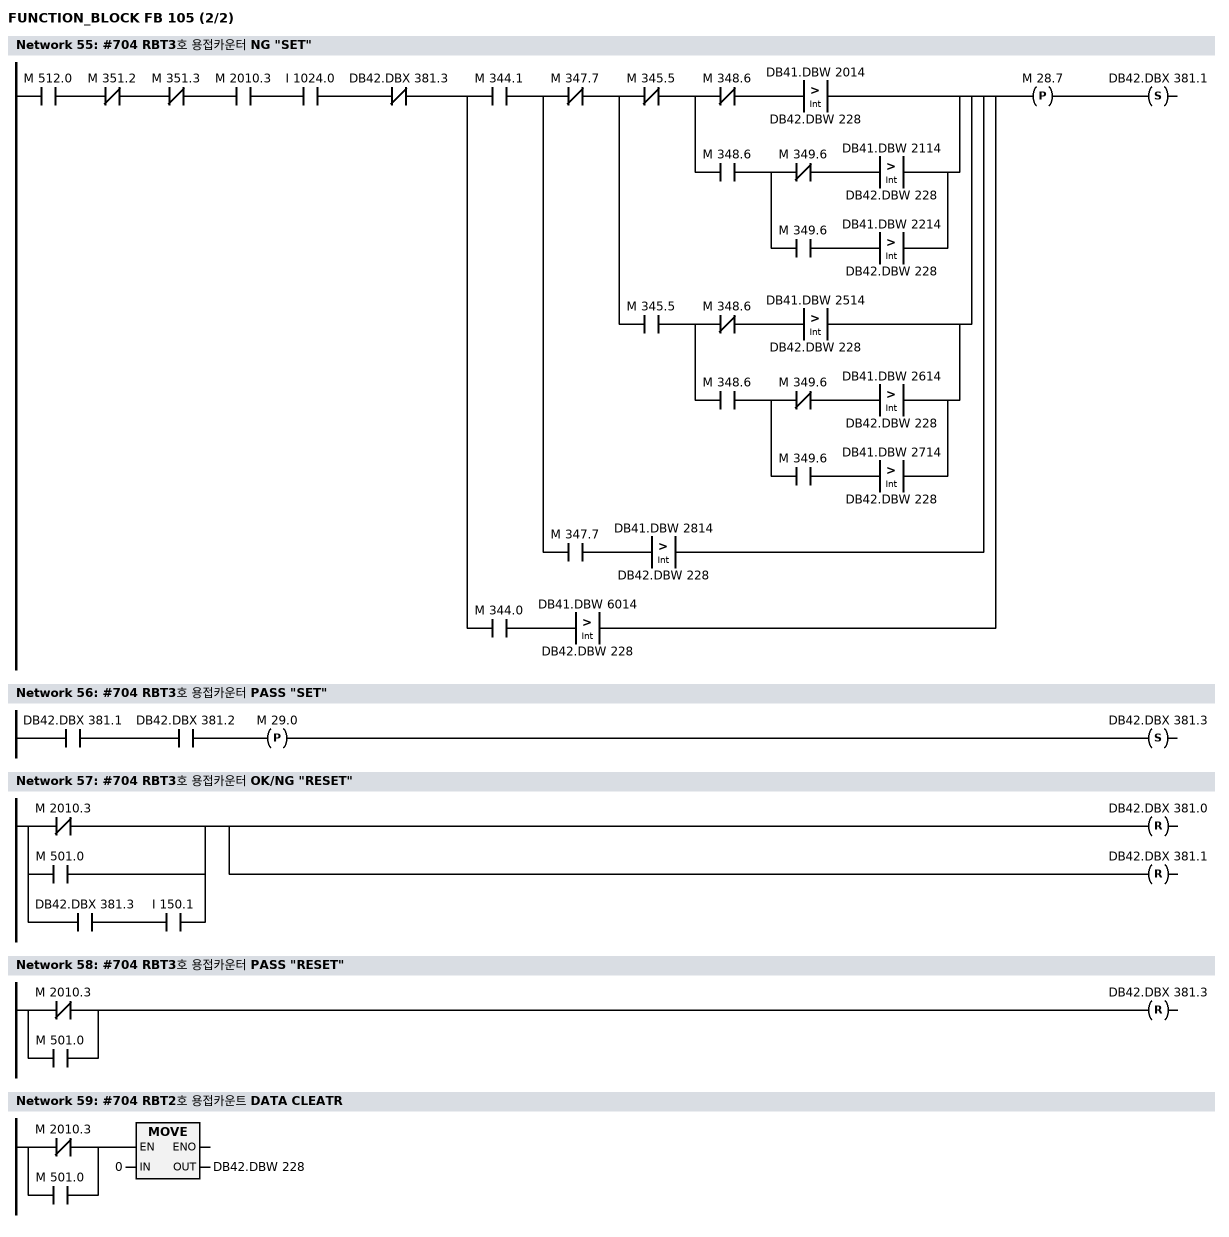

      A     M    512.0;
      AN    M    351.2;
      AN    M    351.3;
      A     M   2010.3;
      A     I   1024.0;
      AN    DB42.DBX  381.3;
      A(    ;
      A     M    344.1;
      A(    ;
      AN    M    347.7;
      A(    ;
      AN    M    345.5;
      A(    ;
      AN    M    348.6;
      A(    ;
      L     DB41.DBW 2014;
      L     DB42.DBW  228;
      >I    ;
      )     ;
      O     ;
      A     M    348.6;
      A(    ;
      AN    M    349.6;
      A(    ;
      L     DB41.DBW 2114;
      L     DB42.DBW  228;
      >I    ;
      )     ;
      O     ;
      A     M    349.6;
      A(    ;
      L     DB41.DBW 2214;
      L     DB42.DBW  228;
      >I    ;
      )     ;
      )     ;
      )     ;
      O     ;
      A     M    345.5;
      A(    ;
      AN    M    348.6;
      A(    ;
      L     DB41.DBW 2514;
      L     DB42.DBW  228;
      >I    ;
      )     ;
      O     ;
      A     M    348.6;
      A(    ;
      AN    M    349.6;
      A(    ;
      L     DB41.DBW 2614;
      L     DB42.DBW  228;
      >I    ;
      )     ;
      O     ;
      A     M    349.6;
      A(    ;
      L     DB41.DBW 2714;
      L     DB42.DBW  228;
      >I    ;
      )     ;
      )     ;
      )     ;
      )     ;
      O     ;
      A     M    347.7;
      A(    ;
      L     DB41.DBW 2814;
      L     DB42.DBW  228;
      >I    ;
      )     ;
      )     ;
      O     ;
      A     M    344.0;
      A(    ;
      L     DB41.DBW 6014;
      L     DB42.DBW  228;
      >I    ;
      )     ;
      )     ;
      FP    M     28.7;
      S     DB42.DBX  381.1;
NETWORK
TITLE =#704 RBT3호 용접카운터 PASS "SET"
//
//
      A     DB42.DBX  381.1;
      A     DB42.DBX  381.2;
      FP    M     29.0;
      S     DB42.DBX  381.3;
NETWORK
TITLE =#704 RBT3호 용접카운터 OK/NG "RESET"

      ON    M   2010.3;
      O     M    501.0;
      O     ;
      A     DB42.DBX  381.3;
      A     I    150.1;
      R     DB42.DBX  381.0;
      R     DB42.DBX  381.1;
NETWORK
TITLE =#704 RBT3호 용접카운터 PASS "RESET"

      ON    M   2010.3;
      O     M    501.0;
      R     DB42.DBX  381.3;
NETWORK
TITLE =#704 RBT2호 용접카운트 DATA CLEATR

      A(    ;
      ON    M   2010.3;
      O     M    501.0;
      )     ;
      JNB   _054;
      L     0;
      T     DB42.DBW  228;
_054: NOP   0;
NETWORK
TITLE =#704 RBT4호 용접카운터 INT -> DB로 전송보조

      AN    OV;
      =     L      2.0;
      A     L      2.0;
      A     I   1036.0;
      =     M     24.0;
      A     L      2.0;
      A     I   1036.1;
      =     M     24.1;
      A     L      2.0;
      A     I   1036.2;
      =     M     24.2;
      A     L      2.0;
      A     I   1036.3;
      =     M     24.3;
      A     L      2.0;
      A     I   1036.4;
      =     M     24.4;
      A     L      2.0;
      AN    M      3.3;
      =     L      2.1;
      A     L      2.1;
      A     I   1036.5;
      =     M     24.5;
      A     L      2.1;
      A     I   1036.6;
      =     M     24.6;
      A     L      2.1;
      A     I   1036.7;
      =     M     24.7;
NETWORK
TITLE =#704 RBT4호 용접카운터 INT -> DB로 전송
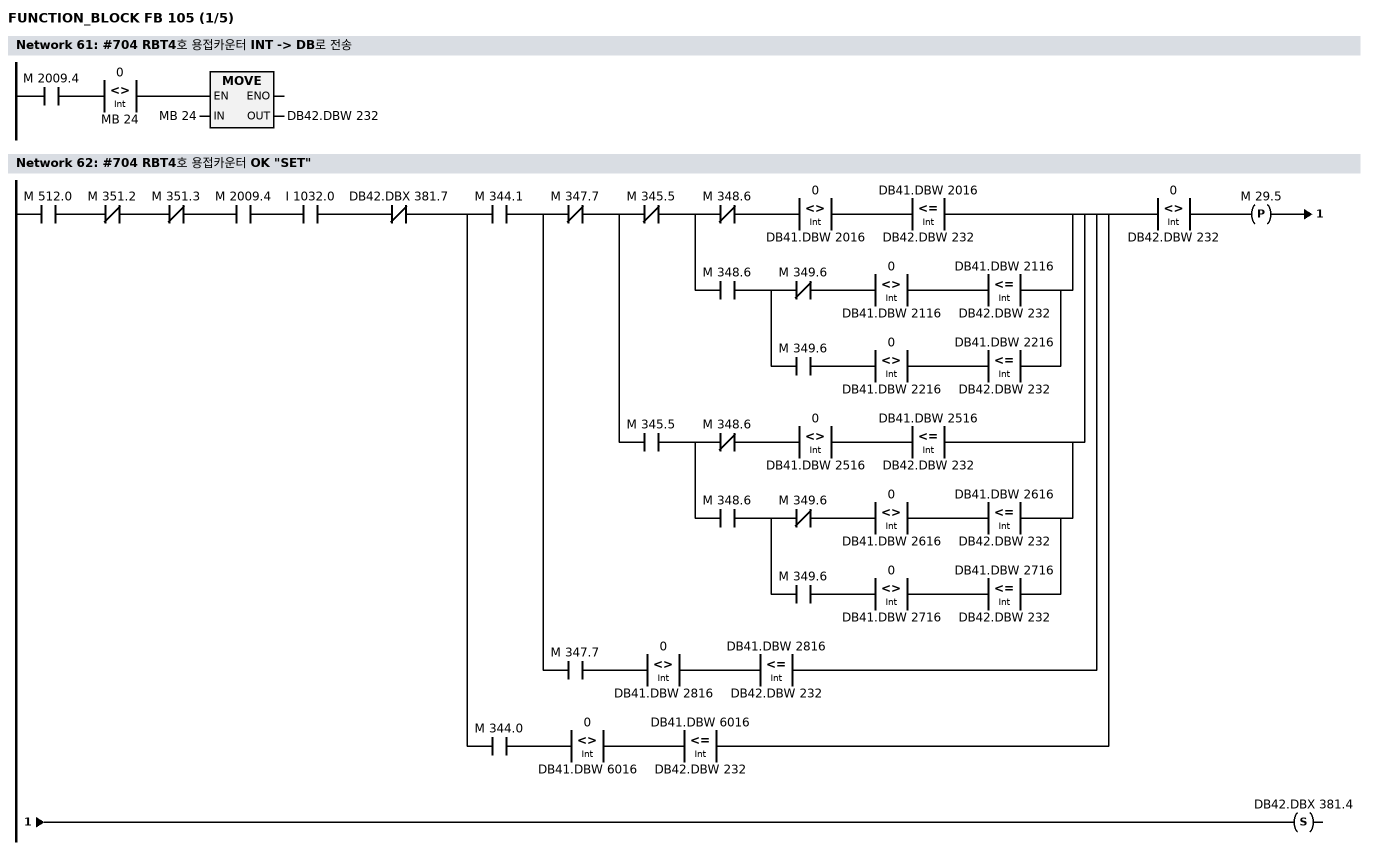

      A     M   2009.4;
      A(    ;
      L     0;
      L     MB    24;
      <>I   ;
      )     ;
      JNB   _055;
      L     MB    24;
      T     DB42.DBW  232;
_055: NOP   0;
NETWORK
TITLE =#704 RBT4호 용접카운터 OK "SET"

      A     M    512.0;
      AN    M    351.2;
      AN    M    351.3;
      A     M   2009.4;
      A     I   1032.0;
      AN    DB42.DBX  381.7;
      A(    ;
      A     M    344.1;
      A(    ;
      AN    M    347.7;
      A(    ;
      AN    M    345.5;
      A(    ;
      AN    M    348.6;
      A(    ;
      L     0;
      L     DB41.DBW 2016;
      <>I   ;
      )     ;
      A(    ;
      L     DB41.DBW 2016;
      L     DB42.DBW  232;
      <=I   ;
      )     ;
      O     ;
      A     M    348.6;
      A(    ;
      AN    M    349.6;
      A(    ;
      L     0;
      L     DB41.DBW 2116;
      <>I   ;
      )     ;
      A(    ;
      L     DB41.DBW 2116;
      L     DB42.DBW  232;
      <=I   ;
      )     ;
      O     ;
      A     M    349.6;
      A(    ;
      L     0;
      L     DB41.DBW 2216;
      <>I   ;
      )     ;
      A(    ;
      L     DB41.DBW 2216;
      L     DB42.DBW  232;
      <=I   ;
      )     ;
      )     ;
      )     ;
      O     ;
      A     M    345.5;
      A(    ;
      AN    M    348.6;
      A(    ;
      L     0;
      L     DB41.DBW 2516;
      <>I   ;
      )     ;
      A(    ;
      L     DB41.DBW 2516;
      L     DB42.DBW  232;
      <=I   ;
      )     ;
      O     ;
      A     M    348.6;
      A(    ;
      AN    M    349.6;
      A(    ;
      L     0;
      L     DB41.DBW 2616;
      <>I   ;
      )     ;
      A(    ;
      L     DB41.DBW 2616;
      L     DB42.DBW  232;
      <=I   ;
      )     ;
      O     ;
      A     M    349.6;
      A(    ;
      L     0;
      L     DB41.DBW 2716;
      <>I   ;
      )     ;
      A(    ;
      L     DB41.DBW 2716;
      L     DB42.DBW  232;
      <=I   ;
      )     ;
      )     ;
      )     ;
      )     ;
      O     ;
      A     M    347.7;
      A(    ;
      L     0;
      L     DB41.DBW 2816;
      <>I   ;
      )     ;
      A(    ;
      L     DB41.DBW 2816;
      L     DB42.DBW  232;
      <=I   ;
      )     ;
      )     ;
      O     ;
      A     M    344.0;
      A(    ;
      L     0;
      L     DB41.DBW 6016;
      <>I   ;
      )     ;
      A(    ;
      L     DB41.DBW 6016;
      L     DB42.DBW  232;
      <=I   ;
      )     ;
      )     ;
      A(    ;
      L     0;
      L     DB42.DBW  232;
      <>I   ;
      )     ;
      FP    M     29.5;
      S     DB42.DBX  381.4;
NETWORK
TITLE =#704 RBT4호 용접카운터 NG "SET"
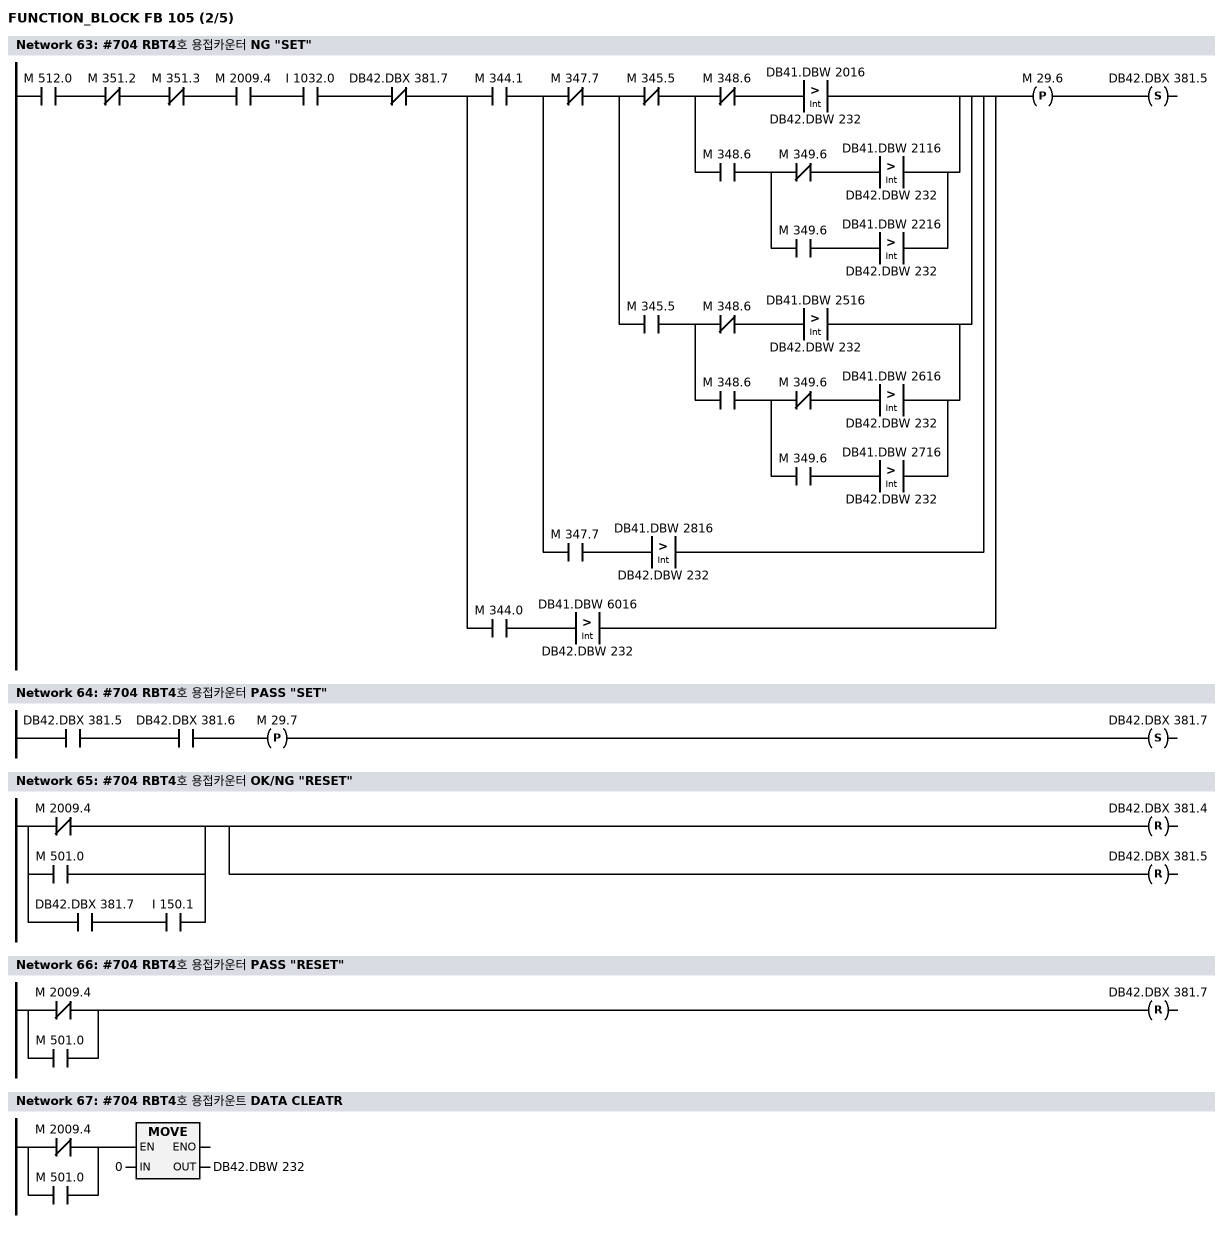

      A     M    512.0;
      AN    M    351.2;
      AN    M    351.3;
      A     M   2009.4;
      A     I   1032.0;
      AN    DB42.DBX  381.7;
      A(    ;
      A     M    344.1;
      A(    ;
      AN    M    347.7;
      A(    ;
      AN    M    345.5;
      A(    ;
      AN    M    348.6;
      A(    ;
      L     DB41.DBW 2016;
      L     DB42.DBW  232;
      >I    ;
      )     ;
      O     ;
      A     M    348.6;
      A(    ;
      AN    M    349.6;
      A(    ;
      L     DB41.DBW 2116;
      L     DB42.DBW  232;
      >I    ;
      )     ;
      O     ;
      A     M    349.6;
      A(    ;
      L     DB41.DBW 2216;
      L     DB42.DBW  232;
      >I    ;
      )     ;
      )     ;
      )     ;
      O     ;
      A     M    345.5;
      A(    ;
      AN    M    348.6;
      A(    ;
      L     DB41.DBW 2516;
      L     DB42.DBW  232;
      >I    ;
      )     ;
      O     ;
      A     M    348.6;
      A(    ;
      AN    M    349.6;
      A(    ;
      L     DB41.DBW 2616;
      L     DB42.DBW  232;
      >I    ;
      )     ;
      O     ;
      A     M    349.6;
      A(    ;
      L     DB41.DBW 2716;
      L     DB42.DBW  232;
      >I    ;
      )     ;
      )     ;
      )     ;
      )     ;
      O     ;
      A     M    347.7;
      A(    ;
      L     DB41.DBW 2816;
      L     DB42.DBW  232;
      >I    ;
      )     ;
      )     ;
      O     ;
      A     M    344.0;
      A(    ;
      L     DB41.DBW 6016;
      L     DB42.DBW  232;
      >I    ;
      )     ;
      )     ;
      FP    M     29.6;
      S     DB42.DBX  381.5;
NETWORK
TITLE =#704 RBT4호 용접카운터 PASS "SET"
//
//
      A     DB42.DBX  381.5;
      A     DB42.DBX  381.6;
      FP    M     29.7;
      S     DB42.DBX  381.7;
NETWORK
TITLE =#704 RBT4호 용접카운터 OK/NG "RESET"

      ON    M   2009.4;
      O     M    501.0;
      O     ;
      A     DB42.DBX  381.7;
      A     I    150.1;
      R     DB42.DBX  381.4;
      R     DB42.DBX  381.5;
NETWORK
TITLE =#704 RBT4호 용접카운터 PASS "RESET"

      ON    M   2009.4;
      O     M    501.0;
      R     DB42.DBX  381.7;
NETWORK
TITLE =#704 RBT4호 용접카운트 DATA CLEATR

      A(    ;
      ON    M   2009.4;
      O     M    501.0;
      )     ;
      JNB   _056;
      L     0;
      T     DB42.DBW  232;
_056: NOP   0;
NETWORK
TITLE =
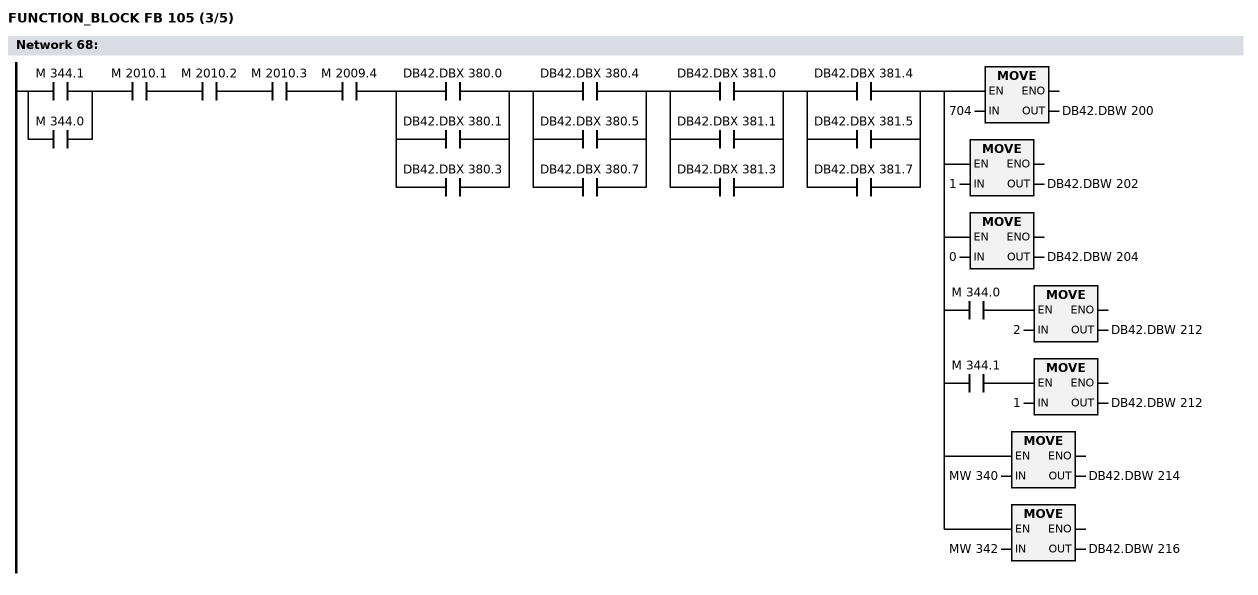

      A(    ;
      O     M    344.1;
      O     M    344.0;
      )     ;
      A     M   2010.1;
      A     M   2010.2;
      A     M   2010.3;
      A     M   2009.4;
      A(    ;
      O     DB42.DBX  380.0;
      O     DB42.DBX  380.1;
      O     DB42.DBX  380.3;
      )     ;
      A(    ;
      O     DB42.DBX  380.4;
      O     DB42.DBX  380.5;
      O     DB42.DBX  380.7;
      )     ;
      A(    ;
      O     DB42.DBX  381.0;
      O     DB42.DBX  381.1;
      O     DB42.DBX  381.3;
      )     ;
      A(    ;
      O     DB42.DBX  381.4;
      O     DB42.DBX  381.5;
      O     DB42.DBX  381.7;
      )     ;
      =     L      2.0;
      A     L      2.0;
      JNB   _057;
      L     704;
      T     DB42.DBW  200;
_057: NOP   0;
      A     L      2.0;
      JNB   _058;
      L     1;
      T     DB42.DBW  202;
_058: NOP   0;
      A     L      2.0;
      JNB   _059;
      L     0;
      T     DB42.DBW  204;
_059: NOP   0;
      A     L      2.0;
      A     M    344.0;
      JNB   _05a;
      L     2;
      T     DB42.DBW  212;
_05a: NOP   0;
      A     L      2.0;
      A     M    344.1;
      JNB   _05b;
      L     1;
      T     DB42.DBW  212;
_05b: NOP   0;
      A     L      2.0;
      JNB   _05c;
      L     MW   340;
      T     DB42.DBW  214;
_05c: NOP   0;
      A     L      2.0;
      JNB   _05d;
      L     MW   342;
      T     DB42.DBW  216;
_05d: NOP   0;
NETWORK
TITLE =
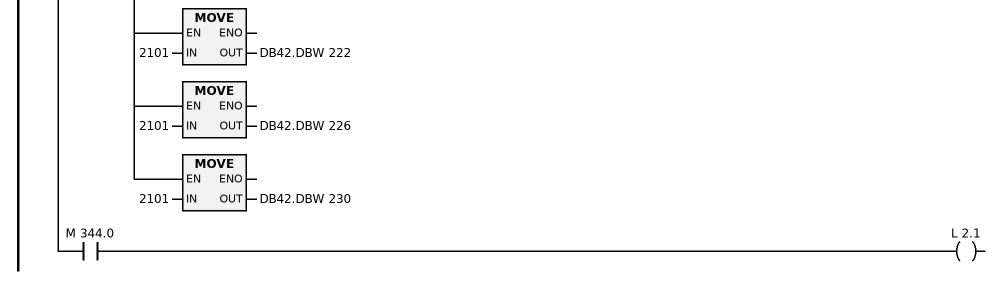

      A(    ;
      O     M    344.1;
      O     M    344.0;
      )     ;
      A     M   2010.1;
      A     M   2010.2;
      A     M   2010.3;
      A     M   2009.4;
      A(    ;
      O     DB42.DBX  380.0;
      O     DB42.DBX  380.1;
      O     DB42.DBX  380.3;
      )     ;
      A(    ;
      O     DB42.DBX  380.4;
      O     DB42.DBX  380.5;
      O     DB42.DBX  380.7;
      )     ;
      A(    ;
      O     DB42.DBX  381.0;
      O     DB42.DBX  381.1;
      O     DB42.DBX  381.3;
      )     ;
      A(    ;
      O     DB42.DBX  381.4;
      O     DB42.DBX  381.5;
      O     DB42.DBX  381.7;
      )     ;
      =     L      2.0;
      A     L      2.0;
      A     M    344.1;
      =     L      2.1;
      A     L      2.1;
      AN    M    347.7;
      =     L      2.2;
      A     L      2.2;
      AN    M    345.5;
      =     L      2.3;
      A     L      2.3;
      AN    M    348.6;
      =     L      2.4;
      A     L      2.4;
      JNB   _05e;
      L     2011;
      T     DB42.DBW  218;
_05e: NOP   0;
      A     L      2.4;
      JNB   _05f;
      L     2011;
      T     DB42.DBW  222;
_05f: NOP   0;
      A     L      2.4;
      JNB   _060;
      L     2011;
      T     DB42.DBW  226;
_060: NOP   0;
      A     L      2.4;
      JNB   _061;
      L     2011;
      T     DB42.DBW  230;
_061: NOP   0;
      A     L      2.3;
      A     M    348.6;
      =     L      2.4;
      A     L      2.4;
      AN    M    349.6;
      =     L      2.5;
      A     L      2.5;
      JNB   _062;
      L     2012;
      T     DB42.DBW  218;
_062: NOP   0;
      A     L      2.5;
      JNB   _063;
      L     2012;
      T     DB42.DBW  222;
_063: NOP   0;
      A     L      2.5;
      JNB   _064;
      L     2012;
      T     DB42.DBW  226;
_064: NOP   0;
      A     L      2.5;
      JNB   _065;
      L     2012;
      T     DB42.DBW  230;
_065: NOP   0;
      A     L      2.4;
      A     M    349.6;
      =     L      2.5;
      A     L      2.5;
      JNB   _066;
      L     2013;
      T     DB42.DBW  218;
_066: NOP   0;
      A     L      2.5;
      JNB   _067;
      L     2013;
      T     DB42.DBW  222;
_067: NOP   0;
      A     L      2.5;
      JNB   _068;
      L     2013;
      T     DB42.DBW  226;
_068: NOP   0;
      A     L      2.5;
      JNB   _069;
      L     2013;
      T     DB42.DBW  230;
_069: NOP   0;
      A     L      2.2;
      A     M    345.5;
      =     L      2.3;
      A     L      2.3;
      AN    M    348.6;
      =     L      2.4;
      A     L      2.4;
      JNB   _06a;
      L     2016;
      T     DB42.DBW  218;
_06a: NOP   0;
      A     L      2.4;
      JNB   _06b;
      L     2016;
      T     DB42.DBW  222;
_06b: NOP   0;
      A     L      2.4;
      JNB   _06c;
      L     2016;
      T     DB42.DBW  226;
_06c: NOP   0;
      A     L      2.4;
      JNB   _06d;
      L     2016;
      T     DB42.DBW  230;
_06d: NOP   0;
      A     L      2.3;
      A     M    348.6;
      =     L      2.4;
      A     L      2.4;
      AN    M    349.6;
      =     L      2.5;
      A     L      2.5;
      JNB   _06e;
      L     2017;
      T     DB42.DBW  218;
_06e: NOP   0;
      A     L      2.5;
      JNB   _06f;
      L     2017;
      T     DB42.DBW  222;
_06f: NOP   0;
      A     L      2.5;
      JNB   _070;
      L     2017;
      T     DB42.DBW  226;
_070: NOP   0;
      A     L      2.5;
      JNB   _071;
      L     2017;
      T     DB42.DBW  230;
_071: NOP   0;
      A     L      2.4;
      A     M    349.6;
      =     L      2.5;
      A     L      2.5;
      JNB   _072;
      L     2018;
      T     DB42.DBW  218;
_072: NOP   0;
      A     L      2.5;
      JNB   _073;
      L     2018;
      T     DB42.DBW  222;
_073: NOP   0;
      A     L      2.5;
      JNB   _074;
      L     2018;
      T     DB42.DBW  226;
_074: NOP   0;
      A     L      2.5;
      JNB   _075;
      L     2018;
      T     DB42.DBW  230;
_075: NOP   0;
      A     L      2.1;
      A     M    347.7;
      =     L      2.2;
      A     L      2.2;
      JNB   _076;
      L     2019;
      T     DB42.DBW  218;
_076: NOP   0;
      A     L      2.2;
      JNB   _077;
      L     2019;
      T     DB42.DBW  222;
_077: NOP   0;
      A     L      2.2;
      JNB   _078;
      L     2019;
      T     DB42.DBW  226;
_078: NOP   0;
      A     L      2.2;
      JNB   _079;
      L     2019;
      T     DB42.DBW  230;
_079: NOP   0;
      A     L      2.0;
      A     M    344.0;
      =     L      2.1;
      A     L      2.1;
      JNB   _07a;
      L     2101;
      T     DB42.DBW  218;
_07a: NOP   0;
      A     L      2.1;
      JNB   _07b;
      L     2101;
      T     DB42.DBW  222;
_07b: NOP   0;
      A     L      2.1;
      JNB   _07c;
      L     2101;
      T     DB42.DBW  226;
_07c: NOP   0;
      A     L      2.1;
      JNB   _07d;
      L     2101;
      T     DB42.DBW  230;
_07d: NOP   0;
NETWORK
TITLE =
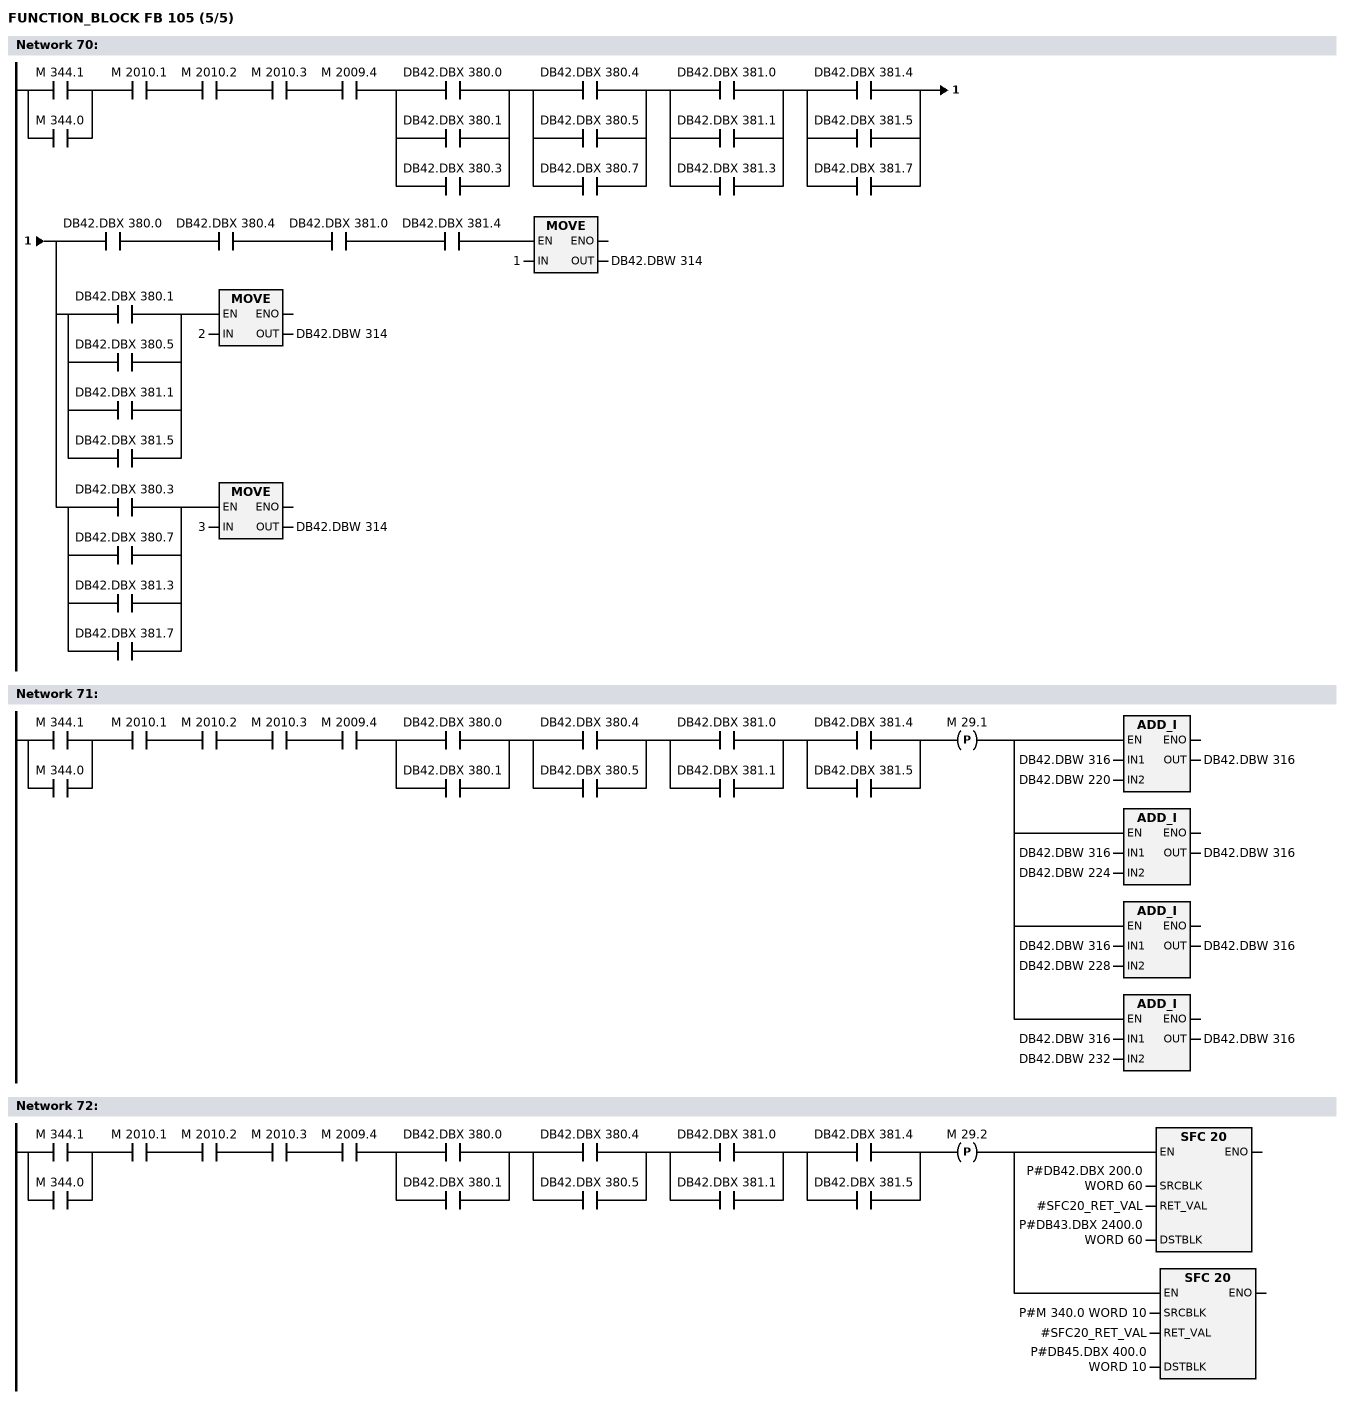

      A(    ;
      O     M    344.1;
      O     M    344.0;
      )     ;
      A     M   2010.1;
      A     M   2010.2;
      A     M   2010.3;
      A     M   2009.4;
      A(    ;
      O     DB42.DBX  380.0;
      O     DB42.DBX  380.1;
      O     DB42.DBX  380.3;
      )     ;
      A(    ;
      O     DB42.DBX  380.4;
      O     DB42.DBX  380.5;
      O     DB42.DBX  380.7;
      )     ;
      A(    ;
      O     DB42.DBX  381.0;
      O     DB42.DBX  381.1;
      O     DB42.DBX  381.3;
      )     ;
      A(    ;
      O     DB42.DBX  381.4;
      O     DB42.DBX  381.5;
      O     DB42.DBX  381.7;
      )     ;
      =     L      2.0;
      A     L      2.0;
      A     DB42.DBX  380.0;
      A     DB42.DBX  380.4;
      A     DB42.DBX  381.0;
      A     DB42.DBX  381.4;
      JNB   _07e;
      L     1;
      T     DB42.DBW  314;
_07e: NOP   0;
      A     L      2.0;
      A(    ;
      O     DB42.DBX  380.1;
      O     DB42.DBX  380.5;
      O     DB42.DBX  381.1;
      O     DB42.DBX  381.5;
      )     ;
      JNB   _07f;
      L     2;
      T     DB42.DBW  314;
_07f: NOP   0;
      A     L      2.0;
      A(    ;
      O     DB42.DBX  380.3;
      O     DB42.DBX  380.7;
      O     DB42.DBX  381.3;
      O     DB42.DBX  381.7;
      )     ;
      JNB   _080;
      L     3;
      T     DB42.DBW  314;
_080: NOP   0;
NETWORK
TITLE =

      A(    ;
      O     M    344.1;
      O     M    344.0;
      )     ;
      A     M   2010.1;
      A     M   2010.2;
      A     M   2010.3;
      A     M   2009.4;
      A(    ;
      O     DB42.DBX  380.0;
      O     DB42.DBX  380.1;
      )     ;
      A(    ;
      O     DB42.DBX  380.4;
      O     DB42.DBX  380.5;
      )     ;
      A(    ;
      O     DB42.DBX  381.0;
      O     DB42.DBX  381.1;
      )     ;
      A(    ;
      O     DB42.DBX  381.4;
      O     DB42.DBX  381.5;
      )     ;
      FP    M     29.1;
      =     L      2.0;
      A     L      2.0;
      JNB   _081;
      L     DB42.DBW  316;
      L     DB42.DBW  220;
      +I    ;
      T     DB42.DBW  316;
_081: NOP   0;
      A     L      2.0;
      JNB   _082;
      L     DB42.DBW  316;
      L     DB42.DBW  224;
      +I    ;
      T     DB42.DBW  316;
_082: NOP   0;
      A     L      2.0;
      JNB   _083;
      L     DB42.DBW  316;
      L     DB42.DBW  228;
      +I    ;
      T     DB42.DBW  316;
_083: NOP   0;
      A     L      2.0;
      JNB   _084;
      L     DB42.DBW  316;
      L     DB42.DBW  232;
      +I    ;
      T     DB42.DBW  316;
_084: NOP   0;
NETWORK
TITLE =

      A(    ;
      O     M    344.1;
      O     M    344.0;
      )     ;
      A     M   2010.1;
      A     M   2010.2;
      A     M   2010.3;
      A     M   2009.4;
      A(    ;
      O     DB42.DBX  380.0;
      O     DB42.DBX  380.1;
      )     ;
      A(    ;
      O     DB42.DBX  380.4;
      O     DB42.DBX  380.5;
      )     ;
      A(    ;
      O     DB42.DBX  381.0;
      O     DB42.DBX  381.1;
      )     ;
      A(    ;
      O     DB42.DBX  381.4;
      O     DB42.DBX  381.5;
      )     ;
      FP    M     29.2;
      =     L      2.0;
      A     L      2.0;
      JNB   _085;
      CALL SFC   20 (
           SRCBLK                   := P#DB42.DBX 200.0 WORD 60,
           RET_VAL                  := #SFC20_RET_VAL,
           DSTBLK                   := P#DB43.DBX 2400.0 WORD 60);
_085: NOP   0;
      A     L      2.0;
      JNB   _086;
      CALL SFC   20 (
           SRCBLK                   := P#M 340.0 WORD 10,
           RET_VAL                  := #SFC20_RET_VAL,
           DSTBLK                   := P#DB45.DBX 400.0 WORD 10);
_086: NOP   0;
NETWORK
TITLE =

      A     M    501.0;
      FP    M     29.3;
      =     L      2.0;
      A(    ;
      A     L      2.0;
      JNB   _087;
      CALL SFC   20 (
           SRCBLK                   := P#DB43.DBX 3360.0 WORD 60,
           RET_VAL                  := #SFC20_RET_VAL,
           DSTBLK                   := P#DB43.DBX 3480.0 WORD 60);
_087: A     BR;
      )     ;
      JNB   _088;
      CALL SFC   20 (
           SRCBLK                   := P#DB43.DBX 3240.0 WORD 60,
           RET_VAL                  := #SFC20_RET_VAL,
           DSTBLK                   := P#DB43.DBX 3360.0 WORD 60);
_088: NOP   0;
      A(    ;
      A     L      2.0;
      JNB   _089;
      CALL SFC   20 (
           SRCBLK                   := P#DB43.DBX 3120.0 WORD 60,
           RET_VAL                  := #SFC20_RET_VAL,
           DSTBLK                   := P#DB43.DBX 3240.0 WORD 60);
_089: A     BR;
      )     ;
      JNB   _08a;
      CALL SFC   20 (
           SRCBLK                   := P#DB43.DBX 3000.0 WORD 60,
           RET_VAL                  := #SFC20_RET_VAL,
           DSTBLK                   := P#DB43.DBX 3120.0 WORD 60);
_08a: NOP   0;
      A(    ;
      A     L      2.0;
      JNB   _08b;
      CALL SFC   20 (
           SRCBLK                   := P#DB43.DBX 2880.0 WORD 60,
           RET_VAL                  := #SFC20_RET_VAL,
           DSTBLK                   := P#DB43.DBX 3000.0 WORD 60);
_08b: A     BR;
      )     ;
      JNB   _08c;
      CALL SFC   20 (
           SRCBLK                   := P#DB43.DBX 2760.0 WORD 60,
           RET_VAL                  := #SFC20_RET_VAL,
           DSTBLK                   := P#DB43.DBX 2880.0 WORD 60);
_08c: NOP   0;
      A(    ;
      A     L      2.0;
      JNB   _08d;
      CALL SFC   20 (
           SRCBLK                   := P#DB43.DBX 2640.0 WORD 60,
           RET_VAL                  := #SFC20_RET_VAL,
           DSTBLK                   := P#DB43.DBX 2760.0 WORD 60);
_08d: A     BR;
      )     ;
      JNB   _08e;
      CALL SFC   20 (
           SRCBLK                   := P#DB43.DBX 2520.0 WORD 60,
           RET_VAL                  := #SFC20_RET_VAL,
           DSTBLK                   := P#DB43.DBX 2640.0 WORD 60);
_08e: NOP   0;
      A     L      2.0;
      JNB   _08f;
      CALL SFC   20 (
           SRCBLK                   := P#DB43.DBX 2400.0 WORD 60,
           RET_VAL                  := #SFC20_RET_VAL,
           DSTBLK                   := P#DB43.DBX 2520.0 WORD 60);
_08f: NOP   0;
      A     L      2.0;
      JNB   _090;
      CALL SFC   21 (
           BVAL                     := P#M 40.0 WORD 1,
           RET_VAL                  := #SFC20_RET_VAL,
           BLK                      := P#DB43.DBX 2400.0 WORD 60);
_090: NOP   0;
      A(    ;
      A     L      2.0;
      JNB   _091;
      CALL SFC   20 (
           SRCBLK                   := P#DB45.DBX 560.0 WORD 10,
           RET_VAL                  := #SFC20_RET_VAL,
           DSTBLK                   := P#DB45.DBX 580.0 WORD 10);
_091: A     BR;
      )     ;
      JNB   _092;
      CALL SFC   20 (
           SRCBLK                   := P#DB45.DBX 540.0 WORD 10,
           RET_VAL                  := #SFC20_RET_VAL,
           DSTBLK                   := P#DB45.DBX 560.0 WORD 10);
_092: NOP   0;
      A(    ;
      A     L      2.0;
      JNB   _093;
      CALL SFC   20 (
           SRCBLK                   := P#DB45.DBX 520.0 WORD 10,
           RET_VAL                  := #SFC20_RET_VAL,
           DSTBLK                   := P#DB45.DBX 540.0 WORD 10);
_093: A     BR;
      )     ;
      JNB   _094;
      CALL SFC   20 (
           SRCBLK                   := P#DB45.DBX 500.0 WORD 10,
           RET_VAL                  := #SFC20_RET_VAL,
           DSTBLK                   := P#DB45.DBX 520.0 WORD 10);
_094: NOP   0;
      A(    ;
      A     L      2.0;
      JNB   _095;
      CALL SFC   20 (
           SRCBLK                   := P#DB45.DBX 480.0 WORD 10,
           RET_VAL                  := #SFC20_RET_VAL,
           DSTBLK                   := P#DB45.DBX 500.0 WORD 10);
_095: A     BR;
      )     ;
      JNB   _096;
      CALL SFC   20 (
           SRCBLK                   := P#DB45.DBX 460.0 WORD 10,
           RET_VAL                  := #SFC20_RET_VAL,
           DSTBLK                   := P#DB45.DBX 480.0 WORD 10);
_096: NOP   0;
      A(    ;
      A     L      2.0;
      JNB   _097;
      CALL SFC   20 (
           SRCBLK                   := P#DB45.DBX 440.0 WORD 10,
           RET_VAL                  := #SFC20_RET_VAL,
           DSTBLK                   := P#DB45.DBX 460.0 WORD 10);
_097: A     BR;
      )     ;
      JNB   _098;
      CALL SFC   20 (
           SRCBLK                   := P#DB45.DBX 420.0 WORD 10,
           RET_VAL                  := #SFC20_RET_VAL,
           DSTBLK                   := P#DB45.DBX 440.0 WORD 10);
_098: NOP   0;
      A     L      2.0;
      JNB   _099;
      CALL SFC   20 (
           SRCBLK                   := P#DB45.DBX 400.0 WORD 10,
           RET_VAL                  := #SFC20_RET_VAL,
           DSTBLK                   := P#DB45.DBX 420.0 WORD 10);
_099: NOP   0;
      A     L      2.0;
      JNB   _09a;
      CALL SFC   21 (
           BVAL                     := P#M 40.0 WORD 1,
           RET_VAL                  := #SFC20_RET_VAL,
           BLK                      := P#DB45.DBX 400.0 WORD 10);
_09a: NOP   0;
NETWORK
TITLE =
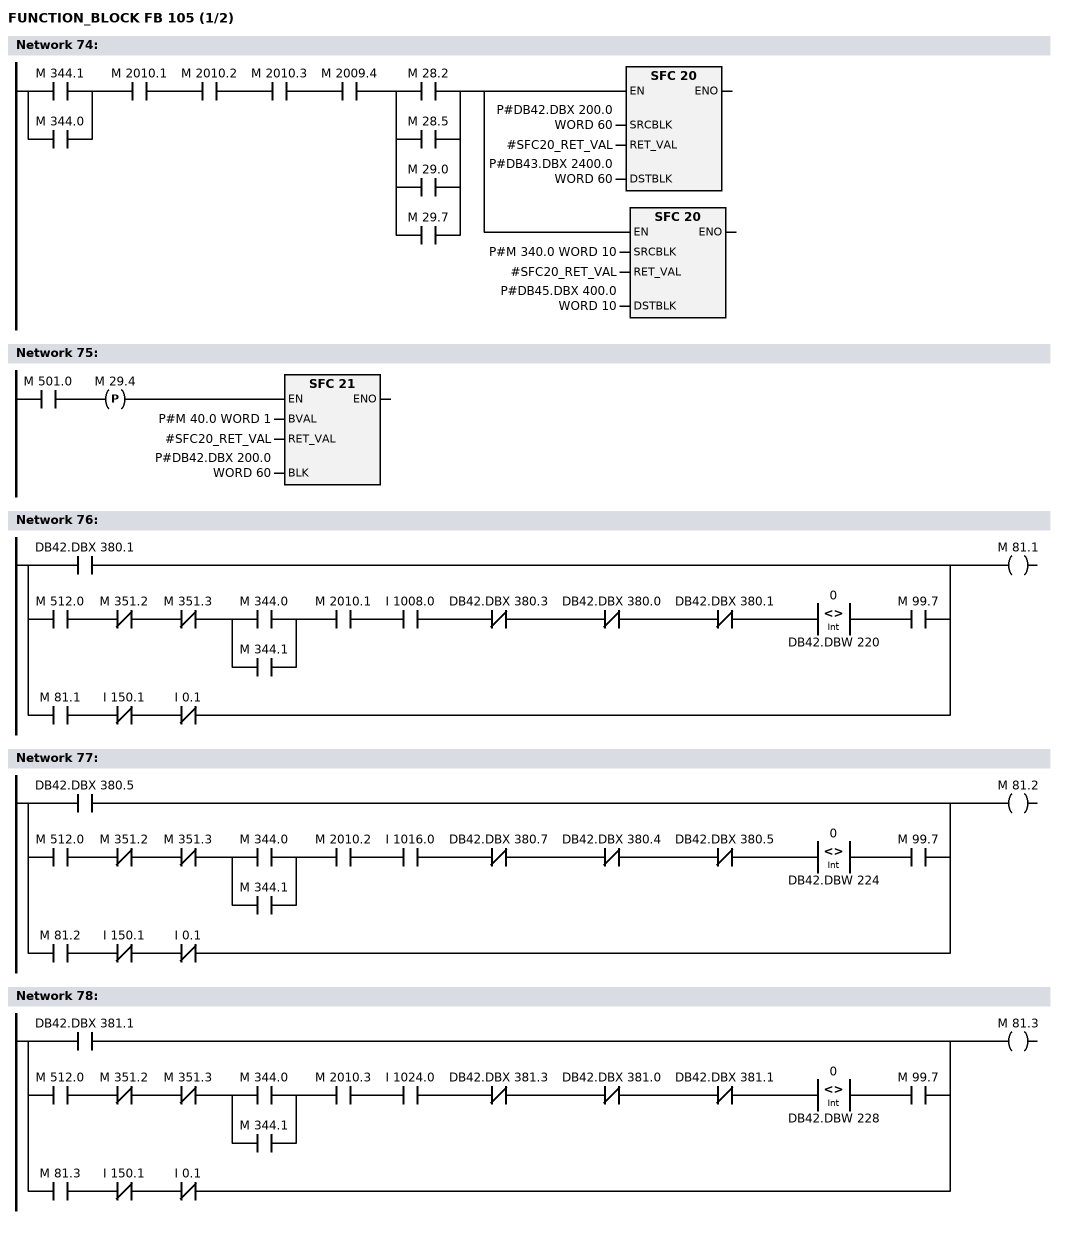

      A(    ;
      O     M    344.1;
      O     M    344.0;
      )     ;
      A     M   2010.1;
      A     M   2010.2;
      A     M   2010.3;
      A     M   2009.4;
      A(    ;
      O     M     28.2;
      O     M     28.5;
      O     M     29.0;
      O     M     29.7;
      )     ;
      =     L      2.0;
      A     L      2.0;
      JNB   _09b;
      CALL SFC   20 (
           SRCBLK                   := P#DB42.DBX 200.0 WORD 60,
           RET_VAL                  := #SFC20_RET_VAL,
           DSTBLK                   := P#DB43.DBX 2400.0 WORD 60);
_09b: NOP   0;
      A     L      2.0;
      JNB   _09c;
      CALL SFC   20 (
           SRCBLK                   := P#M 340.0 WORD 10,
           RET_VAL                  := #SFC20_RET_VAL,
           DSTBLK                   := P#DB45.DBX 400.0 WORD 10);
_09c: NOP   0;
NETWORK
TITLE =

      A     M    501.0;
      FP    M     29.4;
      JNB   _09d;
      CALL SFC   21 (
           BVAL                     := P#M 40.0 WORD 1,
           RET_VAL                  := #SFC20_RET_VAL,
           BLK                      := P#DB42.DBX 200.0 WORD 60);
_09d: NOP   0;
NETWORK
TITLE =

      O     DB42.DBX  380.1;
      O     ;
      A     M    512.0;
      AN    M    351.2;
      AN    M    351.3;
      A(    ;
      O     M    344.0;
      O     M    344.1;
      )     ;
      A     M   2010.1;
      A     I   1008.0;
      AN    DB42.DBX  380.3;
      AN    DB42.DBX  380.0;
      AN    DB42.DBX  380.1;
      A(    ;
      L     0;
      L     DB42.DBW  220;
      <>I   ;
      )     ;
      A     M     99.7;
      O     ;
      A     M     81.1;
      AN    I    150.1;
      AN    I      0.1;
      =     M     81.1;
NETWORK
TITLE =

      O     DB42.DBX  380.5;
      O     ;
      A     M    512.0;
      AN    M    351.2;
      AN    M    351.3;
      A(    ;
      O     M    344.0;
      O     M    344.1;
      )     ;
      A     M   2010.2;
      A     I   1016.0;
      AN    DB42.DBX  380.7;
      AN    DB42.DBX  380.4;
      AN    DB42.DBX  380.5;
      A(    ;
      L     0;
      L     DB42.DBW  224;
      <>I   ;
      )     ;
      A     M     99.7;
      O     ;
      A     M     81.2;
      AN    I    150.1;
      AN    I      0.1;
      =     M     81.2;
NETWORK
TITLE =

      O     DB42.DBX  381.1;
      O     ;
      A     M    512.0;
      AN    M    351.2;
      AN    M    351.3;
      A(    ;
      O     M    344.0;
      O     M    344.1;
      )     ;
      A     M   2010.3;
      A     I   1024.0;
      AN    DB42.DBX  381.3;
      AN    DB42.DBX  381.0;
      AN    DB42.DBX  381.1;
      A(    ;
      L     0;
      L     DB42.DBW  228;
      <>I   ;
      )     ;
      A     M     99.7;
      O     ;
      A     M     81.3;
      AN    I    150.1;
      AN    I      0.1;
      =     M     81.3;
NETWORK
TITLE =
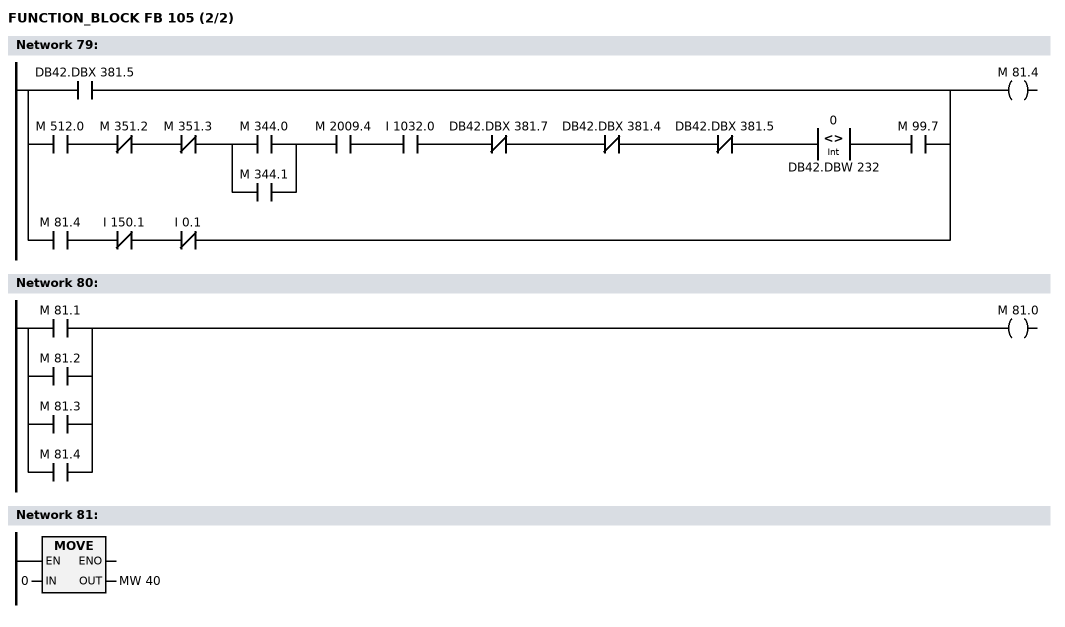

      O     DB42.DBX  381.5;
      O     ;
      A     M    512.0;
      AN    M    351.2;
      AN    M    351.3;
      A(    ;
      O     M    344.0;
      O     M    344.1;
      )     ;
      A     M   2009.4;
      A     I   1032.0;
      AN    DB42.DBX  381.7;
      AN    DB42.DBX  381.4;
      AN    DB42.DBX  381.5;
      A(    ;
      L     0;
      L     DB42.DBW  232;
      <>I   ;
      )     ;
      A     M     99.7;
      O     ;
      A     M     81.4;
      AN    I    150.1;
      AN    I      0.1;
      =     M     81.4;
NETWORK
TITLE =

      O     M     81.1;
      O     M     81.2;
      O     M     81.3;
      O     M     81.4;
      =     M     81.0;
NETWORK
TITLE =

      L     0;
      T     MW    40;
      NOP   0;
END_FUNCTION_BLOCK

DATA_BLOCK DB 105
TITLE =
VERSION : 0.0

 FB 105
BEGIN
   MW_0_BUFF[0] := W#16#0;
   MW_0_BUFF[1] := W#16#0;
   MW_0_BUFF[2] := W#16#0;
   MW_0_BUFF[3] := W#16#0;
   MW_0_BUFF[4] := W#16#0;
   MW_0_BUFF[5] := W#16#0;
   MW_0_BUFF[6] := W#16#0;
   MW_0_BUFF[7] := W#16#0;
   MW_0_BUFF[8] := W#16#0;
   MW_0_BUFF[9] := W#16#0;
   MW_0_BUFF[10] := W#16#0;
   MW_0_BUFF[11] := W#16#0;
   MW_0_BUFF[12] := W#16#0;
   MW_0_BUFF[13] := W#16#0;
   MW_0_BUFF[14] := W#16#0;
   MW_0_BUFF[15] := W#16#0;
   MW_0_BUFF[16] := W#16#0;
   MW_0_BUFF[17] := W#16#0;
   MW_0_BUFF[18] := W#16#0;
   MW_0_BUFF[19] := W#16#0;
   MW_0_BUFF[20] := W#16#0;
   MW_0_BUFF[21] := W#16#0;
   MW_0_BUFF[22] := W#16#0;
   MW_0_BUFF[23] := W#16#0;
   MW_0_BUFF[24] := W#16#0;
   MW_0_BUFF[25] := W#16#0;
   MW_0_BUFF[26] := W#16#0;
   MW_0_BUFF[27] := W#16#0;
   MW_0_BUFF[28] := W#16#0;
   MW_0_BUFF[29] := W#16#0;
   MW_0_BUFF[30] := W#16#0;
   MW_0_BUFF[31] := W#16#0;
   MW_0_BUFF[32] := W#16#0;
   MW_0_BUFF[33] := W#16#0;
   MW_0_BUFF[34] := W#16#0;
   MW_0_BUFF[35] := W#16#0;
   MW_0_BUFF[36] := W#16#0;
   MW_0_BUFF[37] := W#16#0;
   MW_0_BUFF[38] := W#16#0;
   MW_0_BUFF[39] := W#16#0;
   MW_0_BUFF[40] := W#16#0;
   MW_0_BUFF[41] := W#16#0;
   MW_0_BUFF[42] := W#16#0;
   MW_0_BUFF[43] := W#16#0;
   MW_0_BUFF[44] := W#16#0;
   MW_0_BUFF[45] := W#16#0;
   MW_0_BUFF[46] := W#16#0;
   MW_0_BUFF[47] := W#16#0;
   MW_0_BUFF[48] := W#16#0;
   MW_0_BUFF[49] := W#16#0;
   MW_0_BUFF[50] := W#16#0;
   MW_0_BUFF[51] := W#16#0;
   MW_0_BUFF[52] := W#16#0;
   MW_0_BUFF[53] := W#16#0;
   MW_0_BUFF[54] := W#16#0;
   MW_0_BUFF[55] := W#16#0;
   MW_0_BUFF[56] := W#16#0;
   MW_0_BUFF[57] := W#16#0;
   MW_0_BUFF[58] := W#16#0;
   MW_0_BUFF[59] := W#16#0;
   S702_RBT1_WELD_OK_PLS := FALSE;
   S702_RBT1_WELD_NG_PLS := FALSE;
   S702_RBT1_WELD_PASS_PLS := FALSE;
   S702_CHECK_SUM_PLS := FALSE;
   S702_WELD_DATA_MOV_BUFF := FALSE;
   PLS1 := FALSE;
   PLS2 := FALSE;
END_DATA_BLOCK

FUNCTION_BLOCK FB 106
TITLE =
VERSION : 0.1


VAR
  CAR_TYPE_MODIFY : FB 470;
  SFC20_RET_VAL : INT ;
  HMI_CAR_TYPE_V2 : FB 512;
END_VAR
BEGIN
NETWORK
TITLE =
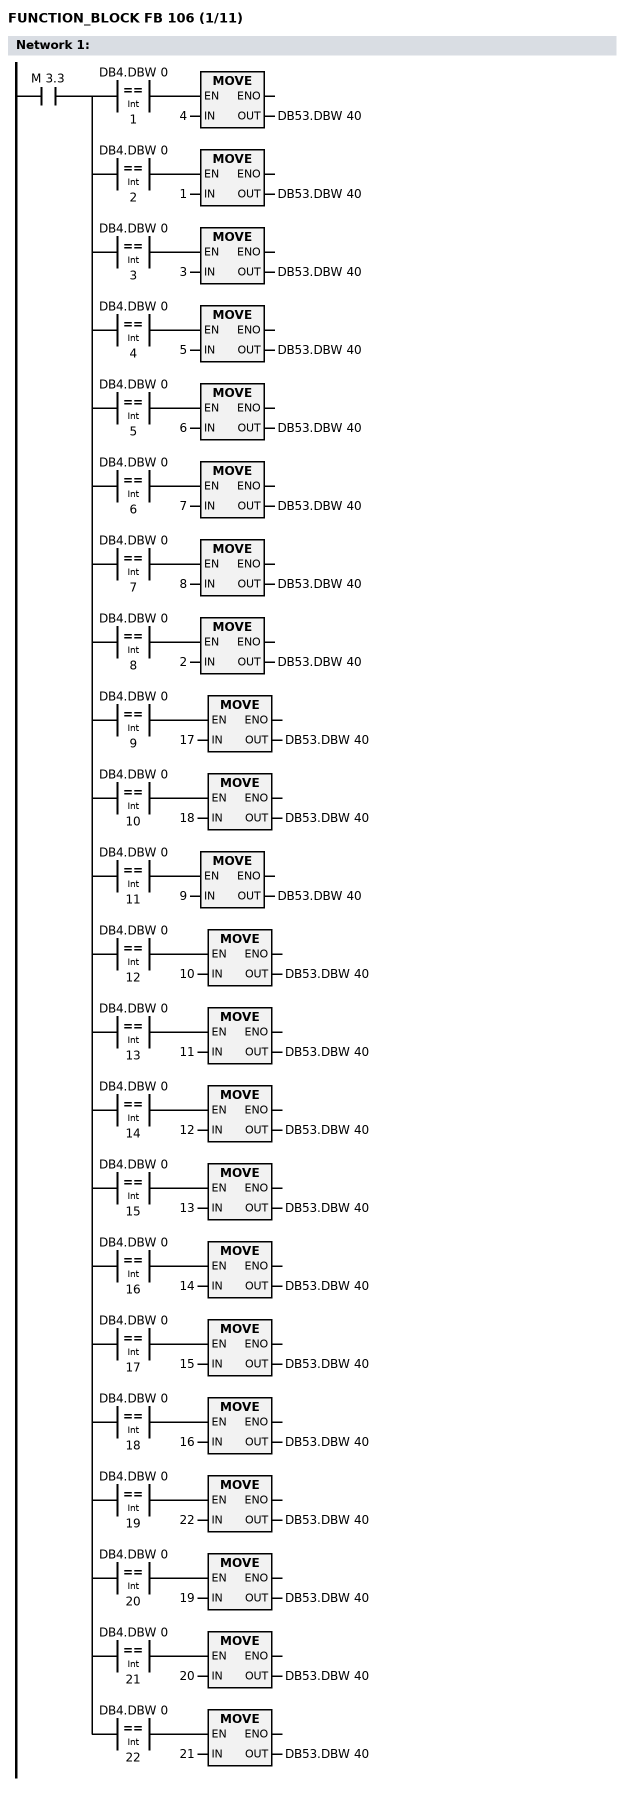

      A     M      3.3;
      =     L      0.0;
      A     L      0.0;
      A(    ;
      L     DB4.DBW    0;
      L     1;
      ==I   ;
      )     ;
      JNB   _001;
      L     4;
      T     DB53.DBW   40;
_001: NOP   0;
      A     L      0.0;
      A(    ;
      L     DB4.DBW    0;
      L     2;
      ==I   ;
      )     ;
      JNB   _002;
      L     1;
      T     DB53.DBW   40;
_002: NOP   0;
      A     L      0.0;
      A(    ;
      L     DB4.DBW    0;
      L     3;
      ==I   ;
      )     ;
      JNB   _003;
      L     3;
      T     DB53.DBW   40;
_003: NOP   0;
      A     L      0.0;
      A(    ;
      L     DB4.DBW    0;
      L     4;
      ==I   ;
      )     ;
      JNB   _004;
      L     5;
      T     DB53.DBW   40;
_004: NOP   0;
      A     L      0.0;
      A(    ;
      L     DB4.DBW    0;
      L     5;
      ==I   ;
      )     ;
      JNB   _005;
      L     6;
      T     DB53.DBW   40;
_005: NOP   0;
      A     L      0.0;
      A(    ;
      L     DB4.DBW    0;
      L     6;
      ==I   ;
      )     ;
      JNB   _006;
      L     7;
      T     DB53.DBW   40;
_006: NOP   0;
      A     L      0.0;
      A(    ;
      L     DB4.DBW    0;
      L     7;
      ==I   ;
      )     ;
      JNB   _007;
      L     8;
      T     DB53.DBW   40;
_007: NOP   0;
      A     L      0.0;
      A(    ;
      L     DB4.DBW    0;
      L     8;
      ==I   ;
      )     ;
      JNB   _008;
      L     2;
      T     DB53.DBW   40;
_008: NOP   0;
      A     L      0.0;
      A(    ;
      L     DB4.DBW    0;
      L     9;
      ==I   ;
      )     ;
      JNB   _009;
      L     17;
      T     DB53.DBW   40;
_009: NOP   0;
      A     L      0.0;
      A(    ;
      L     DB4.DBW    0;
      L     10;
      ==I   ;
      )     ;
      JNB   _00a;
      L     18;
      T     DB53.DBW   40;
_00a: NOP   0;
      A     L      0.0;
      A(    ;
      L     DB4.DBW    0;
      L     11;
      ==I   ;
      )     ;
      JNB   _00b;
      L     9;
      T     DB53.DBW   40;
_00b: NOP   0;
      A     L      0.0;
      A(    ;
      L     DB4.DBW    0;
      L     12;
      ==I   ;
      )     ;
      JNB   _00c;
      L     10;
      T     DB53.DBW   40;
_00c: NOP   0;
      A     L      0.0;
      A(    ;
      L     DB4.DBW    0;
      L     13;
      ==I   ;
      )     ;
      JNB   _00d;
      L     11;
      T     DB53.DBW   40;
_00d: NOP   0;
      A     L      0.0;
      A(    ;
      L     DB4.DBW    0;
      L     14;
      ==I   ;
      )     ;
      JNB   _00e;
      L     12;
      T     DB53.DBW   40;
_00e: NOP   0;
      A     L      0.0;
      A(    ;
      L     DB4.DBW    0;
      L     15;
      ==I   ;
      )     ;
      JNB   _00f;
      L     13;
      T     DB53.DBW   40;
_00f: NOP   0;
      A     L      0.0;
      A(    ;
      L     DB4.DBW    0;
      L     16;
      ==I   ;
      )     ;
      JNB   _010;
      L     14;
      T     DB53.DBW   40;
_010: NOP   0;
      A     L      0.0;
      A(    ;
      L     DB4.DBW    0;
      L     17;
      ==I   ;
      )     ;
      JNB   _011;
      L     15;
      T     DB53.DBW   40;
_011: NOP   0;
      A     L      0.0;
      A(    ;
      L     DB4.DBW    0;
      L     18;
      ==I   ;
      )     ;
      JNB   _012;
      L     16;
      T     DB53.DBW   40;
_012: NOP   0;
      A     L      0.0;
      A(    ;
      L     DB4.DBW    0;
      L     19;
      ==I   ;
      )     ;
      JNB   _013;
      L     22;
      T     DB53.DBW   40;
_013: NOP   0;
      A     L      0.0;
      A(    ;
      L     DB4.DBW    0;
      L     20;
      ==I   ;
      )     ;
      JNB   _014;
      L     19;
      T     DB53.DBW   40;
_014: NOP   0;
      A     L      0.0;
      A(    ;
      L     DB4.DBW    0;
      L     21;
      ==I   ;
      )     ;
      JNB   _015;
      L     20;
      T     DB53.DBW   40;
_015: NOP   0;
      A     L      0.0;
      A(    ;
      L     DB4.DBW    0;
      L     22;
      ==I   ;
      )     ;
      JNB   _016;
      L     21;
      T     DB53.DBW   40;
_016: NOP   0;
NETWORK
TITLE =
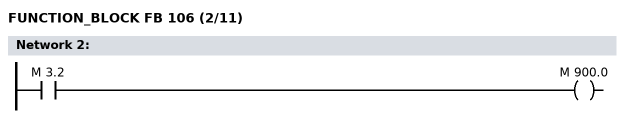

      A     M      3.2;
      =     M    900.0;
NETWORK
TITLE =
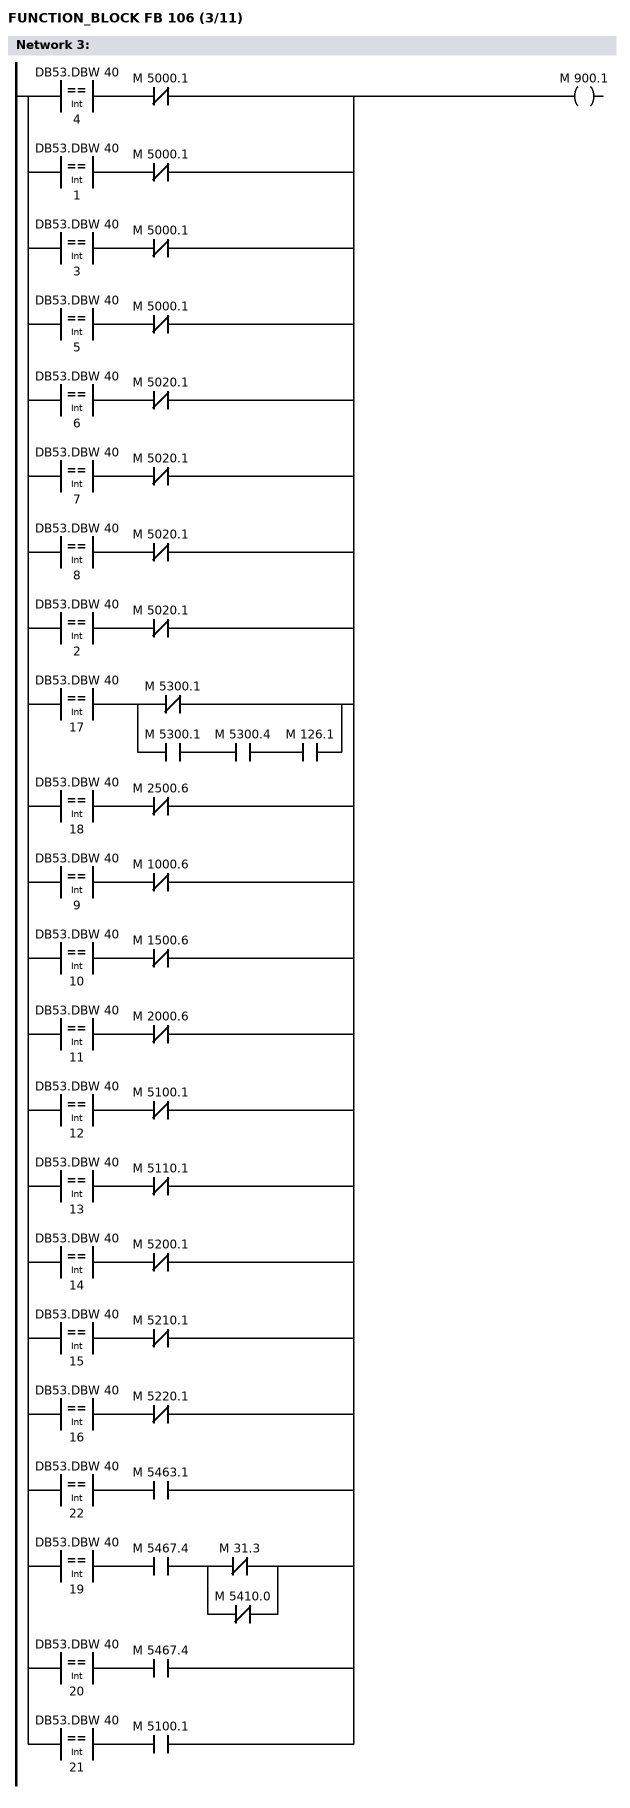

      A(    ;
      L     DB53.DBW   40;
      L     4;
      ==I   ;
      )     ;
      AN    M   5000.1;
      O     ;
      A(    ;
      L     DB53.DBW   40;
      L     1;
      ==I   ;
      )     ;
      AN    M   5000.1;
      O     ;
      A(    ;
      L     DB53.DBW   40;
      L     3;
      ==I   ;
      )     ;
      AN    M   5000.1;
      O     ;
      A(    ;
      L     DB53.DBW   40;
      L     5;
      ==I   ;
      )     ;
      AN    M   5000.1;
      O     ;
      A(    ;
      L     DB53.DBW   40;
      L     6;
      ==I   ;
      )     ;
      AN    M   5020.1;
      O     ;
      A(    ;
      L     DB53.DBW   40;
      L     7;
      ==I   ;
      )     ;
      AN    M   5020.1;
      O     ;
      A(    ;
      L     DB53.DBW   40;
      L     8;
      ==I   ;
      )     ;
      AN    M   5020.1;
      O     ;
      A(    ;
      L     DB53.DBW   40;
      L     2;
      ==I   ;
      )     ;
      AN    M   5020.1;
      O     ;
      A(    ;
      L     DB53.DBW   40;
      L     17;
      ==I   ;
      )     ;
      A(    ;
      ON    M   5300.1;
      O     ;
      A     M   5300.1;
      A     M   5300.4;
      A     M    126.1;
      )     ;
      O     ;
      A(    ;
      L     DB53.DBW   40;
      L     18;
      ==I   ;
      )     ;
      AN    M   2500.6;
      O     ;
      A(    ;
      L     DB53.DBW   40;
      L     9;
      ==I   ;
      )     ;
      AN    M   1000.6;
      O     ;
      A(    ;
      L     DB53.DBW   40;
      L     10;
      ==I   ;
      )     ;
      AN    M   1500.6;
      O     ;
      A(    ;
      L     DB53.DBW   40;
      L     11;
      ==I   ;
      )     ;
      AN    M   2000.6;
      O     ;
      A(    ;
      L     DB53.DBW   40;
      L     12;
      ==I   ;
      )     ;
      AN    M   5100.1;
      O     ;
      A(    ;
      L     DB53.DBW   40;
      L     13;
      ==I   ;
      )     ;
      AN    M   5110.1;
      O     ;
      A(    ;
      L     DB53.DBW   40;
      L     14;
      ==I   ;
      )     ;
      AN    M   5200.1;
      O     ;
      A(    ;
      L     DB53.DBW   40;
      L     15;
      ==I   ;
      )     ;
      AN    M   5210.1;
      O     ;
      A(    ;
      L     DB53.DBW   40;
      L     16;
      ==I   ;
      )     ;
      AN    M   5220.1;
      O     ;
      A(    ;
      L     DB53.DBW   40;
      L     22;
      ==I   ;
      )     ;
      A     M   5463.1;
      O     ;
      A(    ;
      L     DB53.DBW   40;
      L     19;
      ==I   ;
      )     ;
      A     M   5467.4;
      A(    ;
      ON    M     31.3;
      ON    M   5410.0;
      )     ;
      O     ;
      A(    ;
      L     DB53.DBW   40;
      L     20;
      ==I   ;
      )     ;
      A     M   5467.4;
      O     ;
      A(    ;
      L     DB53.DBW   40;
      L     21;
      ==I   ;
      )     ;
      A     M   5100.1;
      =     M    900.1;
NETWORK
TITLE =
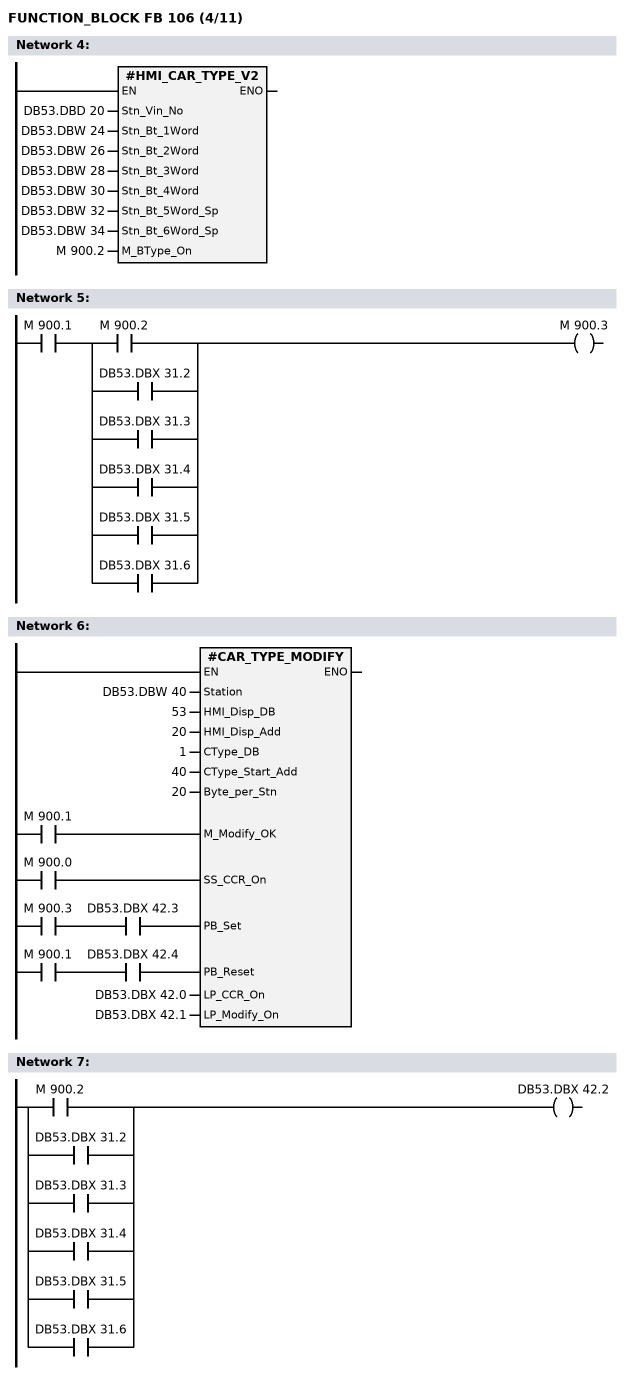

      CALL #HMI_CAR_TYPE_V2 (
           Stn_Vin_No               := DB53.DBD   20,
           Stn_Bt_1Word             := DB53.DBW   24,
           Stn_Bt_2Word             := DB53.DBW   26,
           Stn_Bt_3Word             := DB53.DBW   28,
           Stn_Bt_4Word             := DB53.DBW   30,
           Stn_Bt_5Word_Sp          := DB53.DBW   32,
           Stn_Bt_6Word_Sp          := DB53.DBW   34,
           M_BType_On               := M    900.2);

      NOP   0;
NETWORK
TITLE =

      A     M    900.1;
      A(    ;
      O     M    900.2;
      O     DB53.DBX   31.2;
      O     DB53.DBX   31.3;
      O     DB53.DBX   31.4;
      O     DB53.DBX   31.5;
      O     DB53.DBX   31.6;
      )     ;
      =     M    900.3;
NETWORK
TITLE =

      A     M    900.1;
      =     L      0.0;
      BLD   103;
      A     M    900.0;
      =     L      0.1;
      BLD   103;
      A     M    900.3;
      A     DB53.DBX   42.3;
      =     L      0.2;
      BLD   103;
      A     M    900.1;
      A     DB53.DBX   42.4;
      =     L      0.3;
      BLD   103;
      CALL #CAR_TYPE_MODIFY (
           Station                  := DB53.DBW   40,
           HMI_Disp_DB              := 53,
           HMI_Disp_Add             := 20,
           CType_DB                 := 1,
           CType_Start_Add          := 40,
           Byte_per_Stn             := 20,
           M_Modify_OK              := L      0.0,
           SS_CCR_On                := L      0.1,
           PB_Set                   := L      0.2,
           PB_Reset                 := L      0.3,
           LP_CCR_On                := DB53.DBX   42.0,
           LP_Modify_On             := DB53.DBX   42.1);
      NOP   0;
NETWORK
TITLE =

      O     M    900.2;
      O     DB53.DBX   31.2;
      O     DB53.DBX   31.3;
      O     DB53.DBX   31.4;
      O     DB53.DBX   31.5;
      O     DB53.DBX   31.6;
      =     DB53.DBX   42.2;
NETWORK
TITLE =
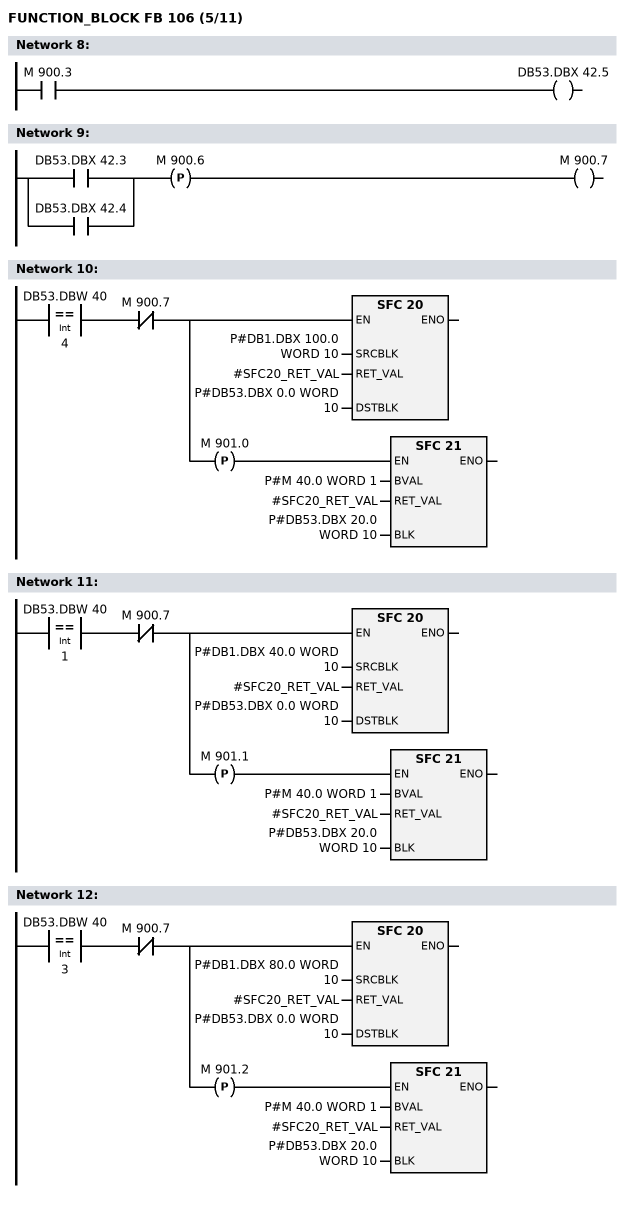

      A     M    900.3;
      =     DB53.DBX   42.5;
NETWORK
TITLE =

      A(    ;
      O     DB53.DBX   42.3;
      O     DB53.DBX   42.4;
      )     ;
      FP    M    900.6;
      =     M    900.7;
NETWORK
TITLE =

      A(    ;
      L     DB53.DBW   40;
      L     4;
      ==I   ;
      )     ;
      AN    M    900.7;
      =     L      0.0;
      A     L      0.0;
      JNB   _017;
      CALL SFC   20 (
           SRCBLK                   := P#DB1.DBX 100.0 WORD 10,
           RET_VAL                  := #SFC20_RET_VAL,
           DSTBLK                   := P#DB53.DBX 0.0 WORD 10);
_017: NOP   0;
      A     L      0.0;
      FP    M    901.0;
      JNB   _018;
      CALL SFC   21 (
           BVAL                     := P#M 40.0 WORD 1,
           RET_VAL                  := #SFC20_RET_VAL,
           BLK                      := P#DB53.DBX 20.0 WORD 10);
_018: NOP   0;
NETWORK
TITLE =

      A(    ;
      L     DB53.DBW   40;
      L     1;
      ==I   ;
      )     ;
      AN    M    900.7;
      =     L      0.0;
      A     L      0.0;
      JNB   _019;
      CALL SFC   20 (
           SRCBLK                   := P#DB1.DBX 40.0 WORD 10,
           RET_VAL                  := #SFC20_RET_VAL,
           DSTBLK                   := P#DB53.DBX 0.0 WORD 10);
_019: NOP   0;
      A     L      0.0;
      FP    M    901.1;
      JNB   _01a;
      CALL SFC   21 (
           BVAL                     := P#M 40.0 WORD 1,
           RET_VAL                  := #SFC20_RET_VAL,
           BLK                      := P#DB53.DBX 20.0 WORD 10);
_01a: NOP   0;
NETWORK
TITLE =

      A(    ;
      L     DB53.DBW   40;
      L     3;
      ==I   ;
      )     ;
      AN    M    900.7;
      =     L      0.0;
      A     L      0.0;
      JNB   _01b;
      CALL SFC   20 (
           SRCBLK                   := P#DB1.DBX 80.0 WORD 10,
           RET_VAL                  := #SFC20_RET_VAL,
           DSTBLK                   := P#DB53.DBX 0.0 WORD 10);
_01b: NOP   0;
      A     L      0.0;
      FP    M    901.2;
      JNB   _01c;
      CALL SFC   21 (
           BVAL                     := P#M 40.0 WORD 1,
           RET_VAL                  := #SFC20_RET_VAL,
           BLK                      := P#DB53.DBX 20.0 WORD 10);
_01c: NOP   0;
NETWORK
TITLE =
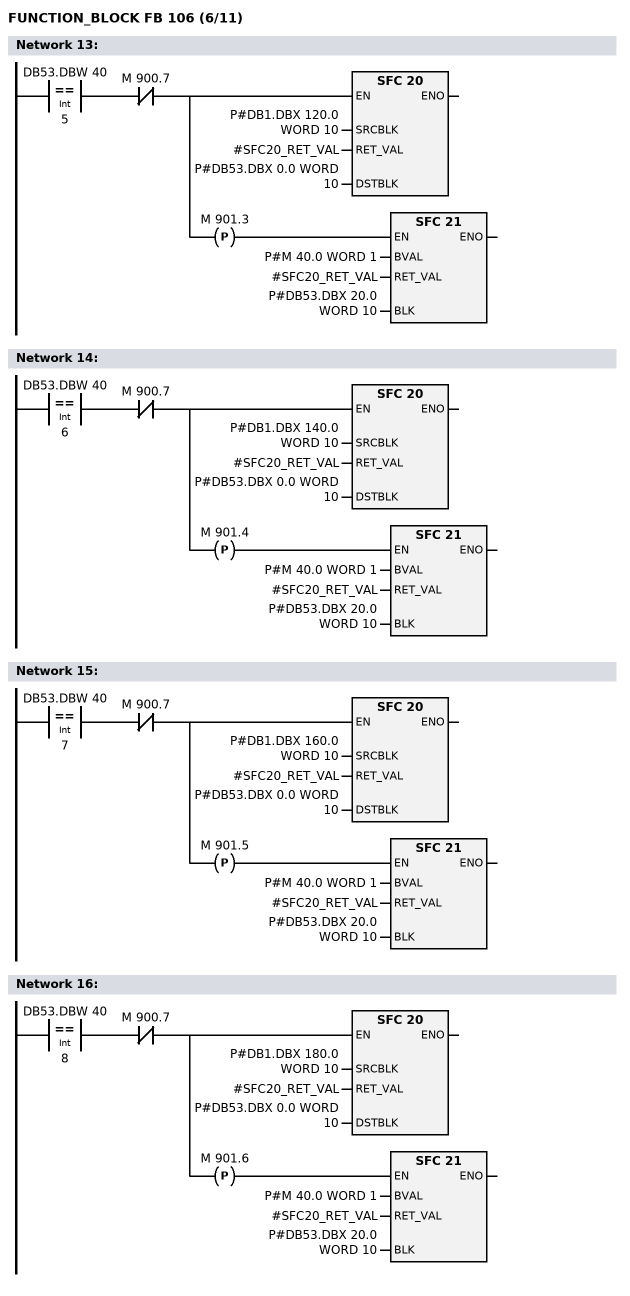

      A(    ;
      L     DB53.DBW   40;
      L     5;
      ==I   ;
      )     ;
      AN    M    900.7;
      =     L      0.0;
      A     L      0.0;
      JNB   _01d;
      CALL SFC   20 (
           SRCBLK                   := P#DB1.DBX 120.0 WORD 10,
           RET_VAL                  := #SFC20_RET_VAL,
           DSTBLK                   := P#DB53.DBX 0.0 WORD 10);
_01d: NOP   0;
      A     L      0.0;
      FP    M    901.3;
      JNB   _01e;
      CALL SFC   21 (
           BVAL                     := P#M 40.0 WORD 1,
           RET_VAL                  := #SFC20_RET_VAL,
           BLK                      := P#DB53.DBX 20.0 WORD 10);
_01e: NOP   0;
NETWORK
TITLE =

      A(    ;
      L     DB53.DBW   40;
      L     6;
      ==I   ;
      )     ;
      AN    M    900.7;
      =     L      0.0;
      A     L      0.0;
      JNB   _01f;
      CALL SFC   20 (
           SRCBLK                   := P#DB1.DBX 140.0 WORD 10,
           RET_VAL                  := #SFC20_RET_VAL,
           DSTBLK                   := P#DB53.DBX 0.0 WORD 10);
_01f: NOP   0;
      A     L      0.0;
      FP    M    901.4;
      JNB   _020;
      CALL SFC   21 (
           BVAL                     := P#M 40.0 WORD 1,
           RET_VAL                  := #SFC20_RET_VAL,
           BLK                      := P#DB53.DBX 20.0 WORD 10);
_020: NOP   0;
NETWORK
TITLE =

      A(    ;
      L     DB53.DBW   40;
      L     7;
      ==I   ;
      )     ;
      AN    M    900.7;
      =     L      0.0;
      A     L      0.0;
      JNB   _021;
      CALL SFC   20 (
           SRCBLK                   := P#DB1.DBX 160.0 WORD 10,
           RET_VAL                  := #SFC20_RET_VAL,
           DSTBLK                   := P#DB53.DBX 0.0 WORD 10);
_021: NOP   0;
      A     L      0.0;
      FP    M    901.5;
      JNB   _022;
      CALL SFC   21 (
           BVAL                     := P#M 40.0 WORD 1,
           RET_VAL                  := #SFC20_RET_VAL,
           BLK                      := P#DB53.DBX 20.0 WORD 10);
_022: NOP   0;
NETWORK
TITLE =

      A(    ;
      L     DB53.DBW   40;
      L     8;
      ==I   ;
      )     ;
      AN    M    900.7;
      =     L      0.0;
      A     L      0.0;
      JNB   _023;
      CALL SFC   20 (
           SRCBLK                   := P#DB1.DBX 180.0 WORD 10,
           RET_VAL                  := #SFC20_RET_VAL,
           DSTBLK                   := P#DB53.DBX 0.0 WORD 10);
_023: NOP   0;
      A     L      0.0;
      FP    M    901.6;
      JNB   _024;
      CALL SFC   21 (
           BVAL                     := P#M 40.0 WORD 1,
           RET_VAL                  := #SFC20_RET_VAL,
           BLK                      := P#DB53.DBX 20.0 WORD 10);
_024: NOP   0;
NETWORK
TITLE =
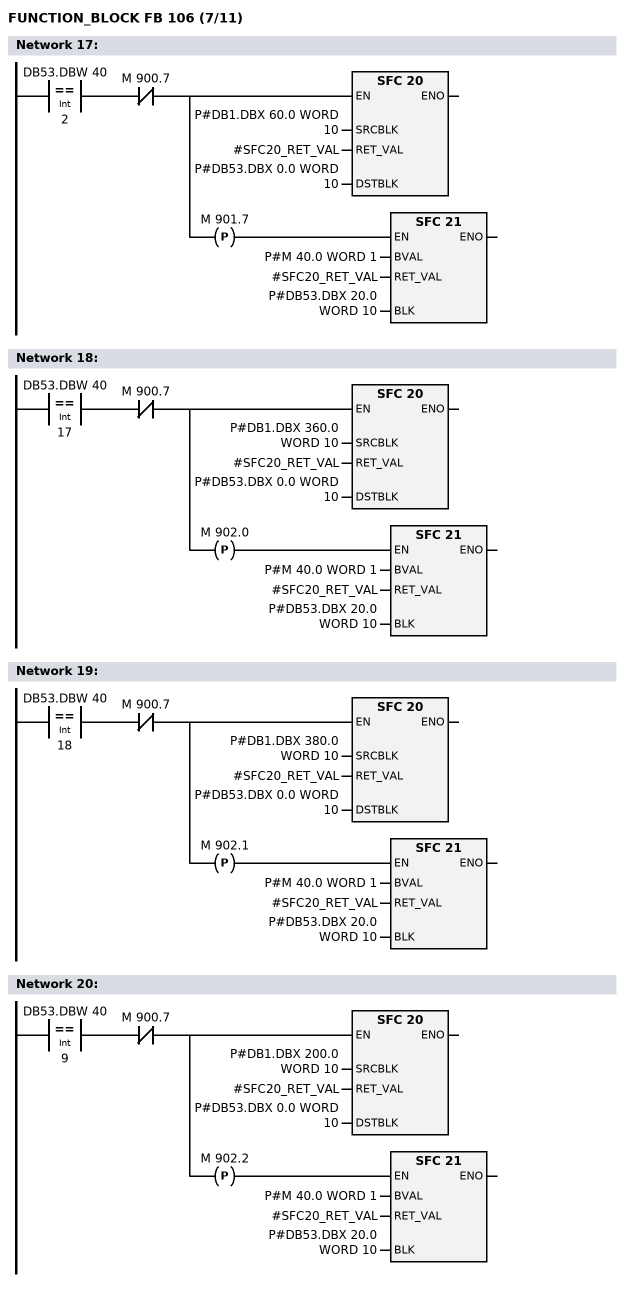

      A(    ;
      L     DB53.DBW   40;
      L     2;
      ==I   ;
      )     ;
      AN    M    900.7;
      =     L      0.0;
      A     L      0.0;
      JNB   _025;
      CALL SFC   20 (
           SRCBLK                   := P#DB1.DBX 60.0 WORD 10,
           RET_VAL                  := #SFC20_RET_VAL,
           DSTBLK                   := P#DB53.DBX 0.0 WORD 10);
_025: NOP   0;
      A     L      0.0;
      FP    M    901.7;
      JNB   _026;
      CALL SFC   21 (
           BVAL                     := P#M 40.0 WORD 1,
           RET_VAL                  := #SFC20_RET_VAL,
           BLK                      := P#DB53.DBX 20.0 WORD 10);
_026: NOP   0;
NETWORK
TITLE =

      A(    ;
      L     DB53.DBW   40;
      L     17;
      ==I   ;
      )     ;
      AN    M    900.7;
      =     L      0.0;
      A     L      0.0;
      JNB   _027;
      CALL SFC   20 (
           SRCBLK                   := P#DB1.DBX 360.0 WORD 10,
           RET_VAL                  := #SFC20_RET_VAL,
           DSTBLK                   := P#DB53.DBX 0.0 WORD 10);
_027: NOP   0;
      A     L      0.0;
      FP    M    902.0;
      JNB   _028;
      CALL SFC   21 (
           BVAL                     := P#M 40.0 WORD 1,
           RET_VAL                  := #SFC20_RET_VAL,
           BLK                      := P#DB53.DBX 20.0 WORD 10);
_028: NOP   0;
NETWORK
TITLE =

      A(    ;
      L     DB53.DBW   40;
      L     18;
      ==I   ;
      )     ;
      AN    M    900.7;
      =     L      0.0;
      A     L      0.0;
      JNB   _029;
      CALL SFC   20 (
           SRCBLK                   := P#DB1.DBX 380.0 WORD 10,
           RET_VAL                  := #SFC20_RET_VAL,
           DSTBLK                   := P#DB53.DBX 0.0 WORD 10);
_029: NOP   0;
      A     L      0.0;
      FP    M    902.1;
      JNB   _02a;
      CALL SFC   21 (
           BVAL                     := P#M 40.0 WORD 1,
           RET_VAL                  := #SFC20_RET_VAL,
           BLK                      := P#DB53.DBX 20.0 WORD 10);
_02a: NOP   0;
NETWORK
TITLE =

      A(    ;
      L     DB53.DBW   40;
      L     9;
      ==I   ;
      )     ;
      AN    M    900.7;
      =     L      0.0;
      A     L      0.0;
      JNB   _02b;
      CALL SFC   20 (
           SRCBLK                   := P#DB1.DBX 200.0 WORD 10,
           RET_VAL                  := #SFC20_RET_VAL,
           DSTBLK                   := P#DB53.DBX 0.0 WORD 10);
_02b: NOP   0;
      A     L      0.0;
      FP    M    902.2;
      JNB   _02c;
      CALL SFC   21 (
           BVAL                     := P#M 40.0 WORD 1,
           RET_VAL                  := #SFC20_RET_VAL,
           BLK                      := P#DB53.DBX 20.0 WORD 10);
_02c: NOP   0;
NETWORK
TITLE =
